LIN {X 0,Y 467.004,Z 300.757,A -85,B 0,C 180,E1 -6622.997,E2 -6622.997} C_VEL
LIN {X 0,Y 470.189,Z 309.996,A -85,B 0,C 180,E1 -6624.811,E2 -6624.811} C_VEL
LIN {X 0,Y 472.686,Z 318.668,A -85,B 0,C 180,E1 -6626.234,E2 -6626.234} C_VEL
LIN {X 0,Y 470.415,Z 339.223,A -85,B 0,C 180,E1 -6628.306,E2 -6628.306} C_VEL
LIN {X 0,Y 473.455,Z 359.975,A -85,B 0,C 180,E1 -6629.227,E2 -6629.227} C_VEL
LIN {X 0,Y 473.986,Z 366.788,A -85,B 0,C 180,E1 -6629.462,E2 -6629.462} C_VEL
LIN {X 0,Y 470.032,Z 462.753,A -85,B 0,C 180,E1 -6631.452,E2 -6631.452} C_VEL
LIN {X 0,Y 467.328,Z 564.491,A -85,B 0,C 180,E1 -6633.396,E2 -6633.396} C_VEL
LIN {X 0,Y 466.49,Z 584.331,A -85,B 0,C 180,E1 -6634.004,E2 -6634.004} C_VEL
LIN {X 0,Y 465.449,Z 603.573,A -85,B 0,C 180,E1 -6634.828,E2 -6634.828} C_VEL
LIN {X 0,Y 464.28,Z 621.738,A -85,B 0,C 180,E1 -6635.847,E2 -6635.847} C_VEL
LIN {X 0,Y 463.025,Z 638.947,A -85,B 0,C 180,E1 -6637.056,E2 -6637.056} C_VEL
LIN {X 0,Y 461.725,Z 655.288,A -85,B 0,C 180,E1 -6638.467,E2 -6638.467} C_VEL
LIN {X 0,Y 460.481,Z 669.969,A -85,B 0,C 180,E1 -6640.003,E2 -6640.003} C_VEL
LIN {X 0,Y 459.311,Z 683.717,A -85,B 0,C 180,E1 -6641.732,E2 -6641.732} C_VEL
LIN {X 0,Y 458.262,Z 696.374,A -85,B 0,C 180,E1 -6643.653,E2 -6643.653} C_VEL
LIN {X 0,Y 457.409,Z 707.461,A -85,B 0,C 180,E1 -6645.7,E2 -6645.7} C_VEL
LIN {X 0,Y 456.77,Z 717.003,A -85,B 0,C 180,E1 -6647.87,E2 -6647.87} C_VEL
LIN {X 0,Y 456.351,Z 724.573,A -85,B 0,C 180,E1 -6650.033,E2 -6650.033} C_VEL
LIN {X 0,Y 456.093,Z 730.779,A -85,B 0,C 180,E1 -6652.315,E2 -6652.315} C_VEL
LIN {X 0,Y 455.974,Z 735.448,A -85,B 0,C 180,E1 -6654.716,E2 -6654.716} C_VEL
LIN {X 0,Y 455.931,Z 738.322,A -85,B 0,C 180,E1 -6657.109,E2 -6657.109} C_VEL
LIN {X 0,Y 455.922,Z 739.49,A -85,B 0,C 180,E1 -6659.498,E2 -6659.498} C_VEL
LIN {X 0,Y 455.92,Z 739.024,A -85,B 0,C 180,E1 -6661.886,E2 -6661.886} C_VEL
LIN {X 0,Y 455.939,Z 736.915,A -85,B 0,C 180,E1 -6664.276,E2 -6664.276} C_VEL
LIN {X 0,Y 456.015,Z 733.052,A -85,B 0,C 180,E1 -6666.674,E2 -6666.674} C_VEL
LIN {X 0,Y 456.209,Z 727.319,A -85,B 0,C 180,E1 -6669.08,E2 -6669.08} C_VEL
LIN {X 0,Y 456.557,Z 720.008,A -85,B 0,C 180,E1 -6671.368,E2 -6671.368} C_VEL
LIN {X 0,Y 457.145,Z 710.687,A -85,B 0,C 180,E1 -6673.664,E2 -6673.664} C_VEL
LIN {X 0,Y 457.968,Z 699.685,A -85,B 0,C 180,E1 -6675.838,E2 -6675.838} C_VEL
LIN {X 0,Y 458.995,Z 687.344,A -85,B 0,C 180,E1 -6677.833,E2 -6677.833} C_VEL
LIN {X 0,Y 460.155,Z 674.019,A -85,B 0,C 180,E1 -6679.616,E2 -6679.616} C_VEL
LIN {X 0,Y 461.415,Z 659.738,A -85,B 0,C 180,E1 -6681.216,E2 -6681.216} C_VEL
LIN {X 0,Y 462.762,Z 643.878,A -85,B 0,C 180,E1 -6682.691,E2 -6682.691} C_VEL
LIN {X 0,Y 464.102,Z 627.202,A -85,B 0,C 180,E1 -6683.961,E2 -6683.961} C_VEL
LIN {X 0,Y 465.366,Z 609.596,A -85,B 0,C 180,E1 -6685.041,E2 -6685.041} C_VEL
LIN {X 0,Y 466.447,Z 591.759,A -85,B 0,C 180,E1 -6685.897,E2 -6685.897} C_VEL
LIN {X 0,Y 467.379,Z 572.839,A -85,B 0,C 180,E1 -6686.571,E2 -6686.571} C_VEL
LIN {X 0,Y 468.043,Z 553.455,A -85,B 0,C 180,E1 -6687.032,E2 -6687.032} C_VEL
LIN {X 0,Y 472.044,Z 364.66,A -85,B 0,C 180,E1 -6690.301,E2 -6690.301} C_VEL
LIN {X 0,Y 468.212,Z 340.667,A -85,B 0,C 180,E1 -6691.092,E2 -6691.092} C_VEL
LIN {X 0,Y 469.992,Z 315.315,A -85,B 0,C 180,E1 -6693.493,E2 -6693.493} C_VEL
LIN {X 0,Y 463.477,Z 296.548,A -85,B 0,C 180,E1 -6696.002,E2 -6696.002} C_VEL
LIN {X 0,Y 457.078,Z 279.761,A -85,B 0,C 180,E1 -6698.464,E2 -6698.464} C_VEL
LIN {X 0,Y 457.07,Z 279.544,A -85,B 0,C 180,E1 -6701.525,E2 -6701.525} C_VEL
LIN {X 0,Y 456.059,Z 279.675,A -85,B 0,C 180,E1 -6702.49,E2 -6702.49} C_VEL
LIN {X 0,Y 449.569,Z 280.487,A -85,B 0,C 180,E1 -6705.278,E2 -6705.278} C_VEL
LIN {X 0,Y 449.122,Z 280.541,A -85,B 0,C 180,E1 -6705.917,E2 -6705.917} C_VEL
LIN {X 0,Y 449.137,Z 280.538,A -85,B 0,C 180,E1 -6709.622,E2 -6709.622} C_VEL
LIN {X 0,Y 449.13,Z 280.537,A -85,B 0,C 180,E1 -6713.37,E2 -6713.37} C_VEL
LIN {X 0,Y 449.119,Z 280.539,A -85,B 0,C 180,E1 -6717.097,E2 -6717.097} C_VEL
LIN {X 0,Y 449.114,Z 280.527,A -85,B 0,C 180,E1 -6720.819,E2 -6720.819} C_VEL
LIN {X 0,Y 449.118,Z 280.528,A -85,B 0,C 180,E1 -6724.552,E2 -6724.552} C_VEL
LIN {X 0,Y 449.137,Z 280.53,A -85,B 0,C 180,E1 -6728.176,E2 -6728.176} C_VEL
LIN {X 0,Y 449.133,Z 280.53,A -85,B 0,C 180,E1 -6731.973,E2 -6731.973} C_VEL
LIN {X 0,Y 449.131,Z 280.608,A -85,B 0,C 180,E1 -6735.752,E2 -6735.752} C_VEL
LIN {X 0,Y 449.544,Z 282.242,A -85,B 0,C 180,E1 -6736.034,E2 -6736.034} C_VEL
LIN {X 0,Y 456.659,Z 302.01,A -85,B 0,C 180,E1 -6738.378,E2 -6738.378} C_VEL
LIN {X 0,Y 460.21,Z 313.576,A -85,B 0,C 180,E1 -6739.673,E2 -6739.673} C_VEL
LIN {X 0,Y 458.853,Z 354.962,A -85,B 0,C 180,E1 -6743.241,E2 -6743.241} C_VEL
LIN {X 0,Y 457.35,Z 396.302,A -85,B 0,C 180,E1 -6746.803,E2 -6746.803} C_VEL
LIN {X 0,Y 455.74,Z 437.908,A -85,B 0,C 180,E1 -6750.376,E2 -6750.376} C_VEL
LIN {X 0,Y 454.421,Z 476.738,A -85,B 0,C 180,E1 -6753.681,E2 -6753.681} C_VEL
LIN {X 0,Y 455.836,Z 490.567,A -85,B 0,C 180,E1 -6753.982,E2 -6753.982} C_VEL
LIN {X 0,Y 454.268,Z 619.633,A -85,B 0,C 180,E1 -6756.087,E2 -6756.087} C_VEL
LIN {X 0,Y 453.856,Z 635.661,A -85,B 0,C 180,E1 -6756.581,E2 -6756.581} C_VEL
LIN {X 0,Y 453.255,Z 650.989,A -85,B 0,C 180,E1 -6757.286,E2 -6757.286} C_VEL
LIN {X 0,Y 452.533,Z 665.232,A -85,B 0,C 180,E1 -6758.169,E2 -6758.169} C_VEL
LIN {X 0,Y 451.63,Z 679.94,A -85,B 0,C 180,E1 -6759.363,E2 -6759.363} C_VEL
LIN {X 0,Y 450.841,Z 692.096,A -85,B 0,C 180,E1 -6760.606,E2 -6760.606} C_VEL
LIN {X 0,Y 450.014,Z 704.083,A -85,B 0,C 180,E1 -6762.144,E2 -6762.144} C_VEL
LIN {X 0,Y 449.336,Z 714.291,A -85,B 0,C 180,E1 -6763.773,E2 -6763.773} C_VEL
LIN {X 0,Y 448.765,Z 723.452,A -85,B 0,C 180,E1 -6765.638,E2 -6765.638} C_VEL
LIN {X 0,Y 448.394,Z 730.619,A -85,B 0,C 180,E1 -6767.518,E2 -6767.518} C_VEL
LIN {X 0,Y 448.159,Z 736.252,A -85,B 0,C 180,E1 -6769.55,E2 -6769.55} C_VEL
LIN {X 0,Y 448.048,Z 740.095,A -85,B 0,C 180,E1 -6771.604,E2 -6771.604} C_VEL
LIN {X 0,Y 448.006,Z 742.118,A -85,B 0,C 180,E1 -6773.684,E2 -6773.684} C_VEL
LIN {X 0,Y 448.004,Z 742.42,A -85,B 0,C 180,E1 -6775.796,E2 -6775.796} C_VEL
LIN {X 0,Y 448.031,Z 741.006,A -85,B 0,C 180,E1 -6777.8,E2 -6777.8} C_VEL
LIN {X 0,Y 448.127,Z 737.586,A -85,B 0,C 180,E1 -6779.984,E2 -6779.984} C_VEL
LIN {X 0,Y 448.31,Z 732.813,A -85,B 0,C 180,E1 -6781.907,E2 -6781.907} C_VEL
LIN {X 0,Y 448.644,Z 726.109,A -85,B 0,C 180,E1 -6783.857,E2 -6783.857} C_VEL
LIN {X 0,Y 449.14,Z 717.93,A -85,B 0,C 180,E1 -6785.678,E2 -6785.678} C_VEL
LIN {X 0,Y 449.832,Z 707.5,A -85,B 0,C 180,E1 -6787.483,E2 -6787.483} C_VEL
LIN {X 0,Y 450.573,Z 696.876,A -85,B 0,C 180,E1 -6788.955,E2 -6788.955} C_VEL
LIN {X 0,Y 451.426,Z 684.129,A -85,B 0,C 180,E1 -6790.365,E2 -6790.365} C_VEL
LIN {X 0,Y 452.278,Z 670.794,A -85,B 0,C 180,E1 -6791.543,E2 -6791.543} C_VEL
LIN {X 0,Y 453.084,Z 656.003,A -85,B 0,C 180,E1 -6792.55,E2 -6792.55} C_VEL
LIN {X 0,Y 453.737,Z 641.285,A -85,B 0,C 180,E1 -6793.308,E2 -6793.308} C_VEL
LIN {X 0,Y 454.202,Z 625.159,A -85,B 0,C 180,E1 -6793.881,E2 -6793.881} C_VEL
LIN {X 0,Y 454.475,Z 607.28,A -85,B 0,C 180,E1 -6794.254,E2 -6794.254} C_VEL
LIN {X 0,Y 455.734,Z 487.115,A -85,B 0,C 180,E1 -6796.2,E2 -6796.2} C_VEL
LIN {X 0,Y 454.494,Z 476.284,A -85,B 0,C 180,E1 -6796.481,E2 -6796.481} C_VEL
LIN {X 0,Y 455.937,Z 434.163,A -85,B 0,C 180,E1 -6800.071,E2 -6800.071} C_VEL
LIN {X 0,Y 457.572,Z 390.761,A -85,B 0,C 180,E1 -6803.766,E2 -6803.766} C_VEL
LIN {X 0,Y 458.845,Z 346.921,A -85,B 0,C 180,E1 -6807.436,E2 -6807.436} C_VEL
LIN {X 0,Y 459.697,Z 311.528,A -85,B 0,C 180,E1 -6810.413,E2 -6810.413} C_VEL
LIN {X 0,Y 453.193,Z 291.764,A -85,B 0,C 180,E1 -6812.612,E2 -6812.612} C_VEL
LIN {X 0,Y 449.163,Z 280.91,A -85,B 0,C 180,E1 -6813.918,E2 -6813.918} C_VEL
LIN {X 0,Y 449.136,Z 280.536,A -85,B 0,C 180,E1 -6814.413,E2 -6814.413} C_VEL
LIN {X 0,Y 449.126,Z 280.539,A -85,B 0,C 180,E1 -6818.174,E2 -6818.174} C_VEL
LIN {X 0,Y 449.102,Z 280.536,A -85,B 0,C 180,E1 -6821.838,E2 -6821.838} C_VEL
LIN {X 0,Y 449.096,Z 280.541,A -85,B 0,C 180,E1 -6825.567,E2 -6825.567} C_VEL
LIN {X 0,Y 449.109,Z 280.539,A -85,B 0,C 180,E1 -6829.221,E2 -6829.221} C_VEL
LIN {X 0,Y 449.141,Z 280.537,A -85,B 0,C 180,E1 -6832.838,E2 -6832.838} C_VEL
LIN {X 0,Y 449.134,Z 280.54,A -85,B 0,C 180,E1 -6836.554,E2 -6836.554} C_VEL
LIN {X 0,Y 449.119,Z 280.544,A -85,B 0,C 180,E1 -6840.255,E2 -6840.255} C_VEL
LIN {X 0,Y 449.103,Z 280.539,A -85,B 0,C 180,E1 -6843.957,E2 -6843.957} C_VEL
LIN {X 0,Y 449.102,Z 280.539,A -85,B 0,C 180,E1 -6847.676,E2 -6847.676} C_VEL
LIN {X 0,Y 449.12,Z 280.538,A -85,B 0,C 180,E1 -6851.298,E2 -6851.298} C_VEL
LIN {X 0,Y 449.142,Z 280.535,A -85,B 0,C 180,E1 -6854.965,E2 -6854.965} C_VEL
LIN {X 0,Y 449.134,Z 280.537,A -85,B 0,C 180,E1 -6858.697,E2 -6858.697} C_VEL
LIN {X 0,Y 449.114,Z 280.538,A -85,B 0,C 180,E1 -6862.376,E2 -6862.376} C_VEL
LIN {X 0,Y 449.104,Z 280.541,A -85,B 0,C 180,E1 -6866.013,E2 -6866.013} C_VEL
LIN {X 0,Y 449.11,Z 280.536,A -85,B 0,C 180,E1 -6869.766,E2 -6869.766} C_VEL
LIN {X 0,Y 449.133,Z 280.537,A -85,B 0,C 180,E1 -6873.406,E2 -6873.406} C_VEL
LIN {X 0,Y 449.139,Z 280.538,A -85,B 0,C 180,E1 -6877.162,E2 -6877.162} C_VEL
LIN {X 0,Y 449.139,Z 280.54,A -85,B 0,C 180,E1 -6880.881,E2 -6880.881} C_VEL
LIN {X 0,Y 449.119,Z 280.541,A -85,B 0,C 180,E1 -6884.572,E2 -6884.572} C_VEL
LIN {X 0,Y 449.141,Z 280.773,A -85,B 0,C 180,E1 -6888.078,E2 -6888.078} C_VEL
LIN {X 0,Y 451.649,Z 287.077,A -85,B 0,C 180,E1 -6889.017,E2 -6889.017} C_VEL
LIN {X 0,Y 460.318,Z 307.995,A -85,B 0,C 180,E1 -6891.841,E2 -6891.841} C_VEL
LIN {X 0,Y 463.887,Z 317.307,A -85,B 0,C 180,E1 -6892.994,E2 -6892.994} C_VEL
LIN {X 0,Y 467.002,Z 323.829,A -85,B 0,C 180,E1 -6893.412,E2 -6893.412} C_VEL
LIN {X 0,Y 469.493,Z 342.184,A -85,B 0,C 180,E1 -6893.988,E2 -6893.988} C_VEL
LIN {X 0,Y 464.853,Z 535.757,A -85,B 0,C 180,E1 -6897.4,E2 -6897.4} C_VEL
LIN {X 0,Y 463.81,Z 578.935,A -85,B 0,C 180,E1 -6898.185,E2 -6898.185} C_VEL
LIN {X 0,Y 462.812,Z 599.678,A -85,B 0,C 180,E1 -6898.776,E2 -6898.776} C_VEL
LIN {X 0,Y 461.518,Z 620.38,A -85,B 0,C 180,E1 -6899.606,E2 -6899.606} C_VEL
LIN {X 0,Y 460.009,Z 640.141,A -85,B 0,C 180,E1 -6900.644,E2 -6900.644} C_VEL
LIN {X 0,Y 458.457,Z 658.206,A -85,B 0,C 180,E1 -6901.827,E2 -6901.827} C_VEL
LIN {X 0,Y 456.739,Z 676.474,A -85,B 0,C 180,E1 -6903.273,E2 -6903.273} C_VEL
LIN {X 0,Y 454.965,Z 694.499,A -85,B 0,C 180,E1 -6904.994,E2 -6904.994} C_VEL
LIN {X 0,Y 453.312,Z 711.029,A -85,B 0,C 180,E1 -6906.885,E2 -6906.885} C_VEL
LIN {X 0,Y 451.875,Z 725.61,A -85,B 0,C 180,E1 -6908.861,E2 -6908.861} C_VEL
LIN {X 0,Y 450.656,Z 738.782,A -85,B 0,C 180,E1 -6910.967,E2 -6910.967} C_VEL
LIN {X 0,Y 449.621,Z 751.154,A -85,B 0,C 180,E1 -6913.331,E2 -6913.331} C_VEL
LIN {X 0,Y 448.858,Z 761.842,A -85,B 0,C 180,E1 -6915.818,E2 -6915.818} C_VEL
LIN {X 0,Y 448.37,Z 770.416,A -85,B 0,C 180,E1 -6918.293,E2 -6918.293} C_VEL
LIN {X 0,Y 448.097,Z 777.147,A -85,B 0,C 180,E1 -6920.757,E2 -6920.757} C_VEL
LIN {X 0,Y 447.976,Z 782.424,A -85,B 0,C 180,E1 -6923.337,E2 -6923.337} C_VEL
LIN {X 0,Y 447.934,Z 785.83,A -85,B 0,C 180,E1 -6925.777,E2 -6925.777} C_VEL
LIN {X 0,Y 447.924,Z 787.706,A -85,B 0,C 180,E1 -6928.339,E2 -6928.339} C_VEL
LIN {X 0,Y 447.93,Z 787.934,A -85,B 0,C 180,E1 -6930.769,E2 -6930.769} C_VEL
LIN {X 0,Y 447.924,Z 786.591,A -85,B 0,C 180,E1 -6933.329,E2 -6933.329} C_VEL
LIN {X 0,Y 447.954,Z 783.781,A -85,B 0,C 180,E1 -6935.766,E2 -6935.766} C_VEL
LIN {X 0,Y 448.055,Z 779.035,A -85,B 0,C 180,E1 -6938.342,E2 -6938.342} C_VEL
LIN {X 0,Y 448.26,Z 772.794,A -85,B 0,C 180,E1 -6940.8,E2 -6940.8} C_VEL
LIN {X 0,Y 448.64,Z 764.715,A -85,B 0,C 180,E1 -6943.272,E2 -6943.272} C_VEL
LIN {X 0,Y 449.278,Z 754.556,A -85,B 0,C 180,E1 -6945.755,E2 -6945.755} C_VEL
LIN {X 0,Y 450.13,Z 743.005,A -85,B 0,C 180,E1 -6948.067,E2 -6948.067} C_VEL
LIN {X 0,Y 451.188,Z 730.06,A -85,B 0,C 180,E1 -6950.226,E2 -6950.226} C_VEL
LIN {X 0,Y 452.465,Z 715.399,A -85,B 0,C 180,E1 -6952.272,E2 -6952.272} C_VEL
LIN {X 0,Y 453.839,Z 699.789,A -85,B 0,C 180,E1 -6954.103,E2 -6954.103} C_VEL
LIN {X 0,Y 455.316,Z 682.894,A -85,B 0,C 180,E1 -6955.774,E2 -6955.774} C_VEL
LIN {X 0,Y 456.751,Z 665.337,A -85,B 0,C 180,E1 -6957.228,E2 -6957.228} C_VEL
LIN {X 0,Y 458.24,Z 646.072,A -85,B 0,C 180,E1 -6958.546,E2 -6958.546} C_VEL
LIN {X 0,Y 459.606,Z 625.931,A -85,B 0,C 180,E1 -6959.656,E2 -6959.656} C_VEL
LIN {X 0,Y 460.785,Z 605.455,A -85,B 0,C 180,E1 -6960.534,E2 -6960.534} C_VEL
LIN {X 0,Y 461.742,Z 584.721,A -85,B 0,C 180,E1 -6961.188,E2 -6961.188} C_VEL
LIN {X 0,Y 462.403,Z 562.319,A -85,B 0,C 180,E1 -6961.658,E2 -6961.658} C_VEL
LIN {X 0,Y 464.451,Z 466.12,A -85,B 0,C 180,E1 -6963.371,E2 -6963.371} C_VEL
LIN {X 0,Y 467.579,Z 374.807,A -85,B 0,C 180,E1 -6965.199,E2 -6965.199} C_VEL
LIN {X 0,Y 468.939,Z 339.731,A -85,B 0,C 180,E1 -6965.974,E2 -6965.974} C_VEL
LIN {X 0,Y 467.087,Z 323.355,A -85,B 0,C 180,E1 -6966.634,E2 -6966.634} C_VEL
LIN {X 0,Y 466.104,Z 320.719,A -85,B 0,C 180,E1 -6966.917,E2 -6966.917} C_VEL
LIN {X 0,Y 463.19,Z 310.793,A -85,B 0,C 180,E1 -6968.51,E2 -6968.51} C_VEL
LIN {X 0,Y 460.486,Z 303.252,A -85,B 0,C 180,E1 -6970.049,E2 -6970.049} C_VEL
LIN {X 0,Y 458.316,Z 298.482,A -85,B 0,C 180,E1 -6971.379,E2 -6971.379} C_VEL
LIN {X 0,Y 456.97,Z 295.312,A -85,B 0,C 180,E1 -6972.493,E2 -6972.493} C_VEL
LIN {X 0,Y 455.479,Z 292.157,A -85,B 0,C 180,E1 -6974.306,E2 -6974.306} C_VEL
LIN {X 0,Y 455.145,Z 291.254,A -85,B 0,C 180,E1 -6975.379,E2 -6975.379} C_VEL
LIN {X 0,Y 455.306,Z 291.516,A -85,B 0,C 180,E1 -6977.097,E2 -6977.097} C_VEL
LIN {X 0,Y 456.358,Z 294.584,A -85,B 0,C 180,E1 -6979.103,E2 -6979.103} C_VEL
LIN {X 0,Y 457.325,Z 296.299,A -85,B 0,C 180,E1 -6979.927,E2 -6979.927} C_VEL
LIN {X 0,Y 458.999,Z 300.428,A -85,B 0,C 180,E1 -6981.305,E2 -6981.305} C_VEL
LIN {X 0,Y 461.244,Z 306.052,A -85,B 0,C 180,E1 -6982.786,E2 -6982.786} C_VEL
LIN {X 0,Y 464.121,Z 314.873,A -85,B 0,C 180,E1 -6984.584,E2 -6984.584} C_VEL
LIN {X 0,Y 466.083,Z 322.779,A -85,B 0,C 180,E1 -6985.901,E2 -6985.901} C_VEL
LIN {X 0,Y 464.085,Z 338.535,A -85,B 0,C 180,E1 -6987.539,E2 -6987.539} C_VEL
LIN {X 0,Y 466.875,Z 358.34,A -85,B 0,C 180,E1 -6988.493,E2 -6988.493} C_VEL
LIN {X 0,Y 467.732,Z 367.877,A -85,B 0,C 180,E1 -6988.866,E2 -6988.866} C_VEL
LIN {X 0,Y 463.358,Z 459.298,A -85,B 0,C 180,E1 -6990.861,E2 -6990.861} C_VEL
LIN {X 0,Y 460.584,Z 549.83,A -85,B 0,C 180,E1 -6992.649,E2 -6992.649} C_VEL
LIN {X 0,Y 459.83,Z 571.487,A -85,B 0,C 180,E1 -6993.154,E2 -6993.154} C_VEL
LIN {X 0,Y 458.842,Z 591.186,A -85,B 0,C 180,E1 -6993.854,E2 -6993.854} C_VEL
LIN {X 0,Y 457.656,Z 610.428,A -85,B 0,C 180,E1 -6994.785,E2 -6994.785} C_VEL
LIN {X 0,Y 456.377,Z 628.154,A -85,B 0,C 180,E1 -6995.884,E2 -6995.884} C_VEL
LIN {X 0,Y 455.03,Z 644.916,A -85,B 0,C 180,E1 -6997.17,E2 -6997.17} C_VEL
LIN {X 0,Y 453.711,Z 660.341,A -85,B 0,C 180,E1 -6998.61,E2 -6998.61} C_VEL
LIN {X 0,Y 452.418,Z 674.823,A -85,B 0,C 180,E1 -7000.237,E2 -7000.237} C_VEL
LIN {X 0,Y 451.209,Z 688.298,A -85,B 0,C 180,E1 -7002.061,E2 -7002.061} C_VEL
LIN {X 0,Y 450.168,Z 700.262,A -85,B 0,C 180,E1 -7004.014,E2 -7004.014} C_VEL
LIN {X 0,Y 449.334,Z 710.752,A -85,B 0,C 180,E1 -7006.095,E2 -7006.095} C_VEL
LIN {X 0,Y 448.713,Z 719.754,A -85,B 0,C 180,E1 -7008.301,E2 -7008.301} C_VEL
LIN {X 0,Y 448.319,Z 726.882,A -85,B 0,C 180,E1 -7010.501,E2 -7010.501} C_VEL
LIN {X 0,Y 448.084,Z 732.617,A -85,B 0,C 180,E1 -7012.822,E2 -7012.822} C_VEL
LIN {X 0,Y 447.975,Z 736.798,A -85,B 0,C 180,E1 -7015.263,E2 -7015.263} C_VEL
LIN {X 0,Y 447.941,Z 739.228,A -85,B 0,C 180,E1 -7017.698,E2 -7017.698} C_VEL
LIN {X 0,Y 447.94,Z 739.996,A -85,B 0,C 180,E1 -7020.128,E2 -7020.128} C_VEL
LIN {X 0,Y 447.94,Z 739.07,A -85,B 0,C 180,E1 -7022.559,E2 -7022.559} C_VEL
LIN {X 0,Y 447.974,Z 736.442,A -85,B 0,C 180,E1 -7024.994,E2 -7024.994} C_VEL
LIN {X 0,Y 448.088,Z 732.064,A -85,B 0,C 180,E1 -7027.437,E2 -7027.437} C_VEL
LIN {X 0,Y 448.35,Z 725.79,A -85,B 0,C 180,E1 -7029.888,E2 -7029.888} C_VEL
LIN {X 0,Y 448.796,Z 717.917,A -85,B 0,C 180,E1 -7032.219,E2 -7032.219} C_VEL
LIN {X 0,Y 449.462,Z 708.514,A -85,B 0,C 180,E1 -7034.428,E2 -7034.428} C_VEL
LIN {X 0,Y 450.354,Z 697.621,A -85,B 0,C 180,E1 -7036.51,E2 -7036.51} C_VEL
LIN {X 0,Y 451.46,Z 685.251,A -85,B 0,C 180,E1 -7038.464,E2 -7038.464} C_VEL
LIN {X 0,Y 452.754,Z 671.351,A -85,B 0,C 180,E1 -7040.287,E2 -7040.287} C_VEL
LIN {X 0,Y 454.128,Z 656.651,A -85,B 0,C 180,E1 -7041.892,E2 -7041.892} C_VEL
LIN {X 0,Y 455.557,Z 640.643,A -85,B 0,C 180,E1 -7043.339,E2 -7043.339} C_VEL
LIN {X 0,Y 456.934,Z 624.078,A -85,B 0,C 180,E1 -7044.568,E2 -7044.568} C_VEL
LIN {X 0,Y 458.211,Z 606.847,A -85,B 0,C 180,E1 -7045.599,E2 -7045.599} C_VEL
LIN {X 0,Y 459.404,Z 587.701,A -85,B 0,C 180,E1 -7046.481,E2 -7046.481} C_VEL
LIN {X 0,Y 460.322,Z 568.448,A -85,B 0,C 180,E1 -7047.124,E2 -7047.124} C_VEL
LIN {X 0,Y 460.979,Z 547.683,A -85,B 0,C 180,E1 -7047.57,E2 -7047.57} C_VEL
LIN {X 0,Y 465.162,Z 367.88,A -85,B 0,C 180,E1 -7050.755,E2 -7050.755} C_VEL
LIN {X 0,Y 464.681,Z 362.556,A -85,B 0,C 180,E1 -7050.899,E2 -7050.899} C_VEL
LIN {X 0,Y 461.179,Z 340.621,A -85,B 0,C 180,E1 -7051.647,E2 -7051.647} C_VEL
LIN {X 0,Y 462.937,Z 318.632,A -85,B 0,C 180,E1 -7053.743,E2 -7053.743} C_VEL
LIN {X 0,Y 456.59,Z 300.164,A -85,B 0,C 180,E1 -7056.247,E2 -7056.247} C_VEL
LIN {X 0,Y 449.169,Z 280.738,A -85,B 0,C 180,E1 -7059.135,E2 -7059.135} C_VEL
LIN {X 0,Y 449.133,Z 280.54,A -85,B 0,C 180,E1 -7062.766,E2 -7062.766} C_VEL
LIN {X 0,Y 449.122,Z 280.541,A -85,B 0,C 180,E1 -7065.917,E2 -7065.917} C_VEL
LIN {X 0,Y 448.112,Z 280.666,A -85,B 0,C 180,E1 -7066.899,E2 -7066.899} C_VEL
LIN {X 0,Y 441.609,Z 281.477,A -85,B 0,C 180,E1 -7069.738,E2 -7069.738} C_VEL
LIN {X 0,Y 441.192,Z 281.529,A -85,B 0,C 180,E1 -7070.388,E2 -7070.388} C_VEL
LIN {X 0,Y 441.191,Z 281.529,A -85,B 0,C 180,E1 -7074.227,E2 -7074.227} C_VEL
LIN {X 0,Y 441.198,Z 281.527,A -85,B 0,C 180,E1 -7077.973,E2 -7077.973} C_VEL
LIN {X 0,Y 441.199,Z 281.519,A -85,B 0,C 180,E1 -7081.728,E2 -7081.728} C_VEL
LIN {X 0,Y 441.18,Z 281.517,A -85,B 0,C 180,E1 -7085.496,E2 -7085.496} C_VEL
LIN {X 0,Y 441.158,Z 281.522,A -85,B 0,C 180,E1 -7089.154,E2 -7089.154} C_VEL
LIN {X 0,Y 441.149,Z 281.531,A -85,B 0,C 180,E1 -7092.863,E2 -7092.863} C_VEL
LIN {X 0,Y 441.173,Z 281.72,A -85,B 0,C 180,E1 -7095.227,E2 -7095.227} C_VEL
LIN {X 0,Y 442.32,Z 284.77,A -85,B 0,C 180,E1 -7095.668,E2 -7095.668} C_VEL
LIN {X 0,Y 450.223,Z 307.11,A -85,B 0,C 180,E1 -7098.347,E2 -7098.347} C_VEL
LIN {X 0,Y 452.973,Z 316.25,A -85,B 0,C 180,E1 -7099.378,E2 -7099.378} C_VEL
LIN {X 0,Y 451.506,Z 357.126,A -85,B 0,C 180,E1 -7102.939,E2 -7102.939} C_VEL
LIN {X 0,Y 449.934,Z 398.081,A -85,B 0,C 180,E1 -7106.495,E2 -7106.495} C_VEL
LIN {X 0,Y 448.236,Z 439.173,A -85,B 0,C 180,E1 -7110.063,E2 -7110.063} C_VEL
LIN {X 0,Y 446.887,Z 477.018,A -85,B 0,C 180,E1 -7113.309,E2 -7113.309} C_VEL
LIN {X 0,Y 448.356,Z 491.357,A -85,B 0,C 180,E1 -7113.631,E2 -7113.631} C_VEL
LIN {X 0,Y 446.695,Z 620.089,A -85,B 0,C 180,E1 -7115.763,E2 -7115.763} C_VEL
LIN {X 0,Y 446.261,Z 636.081,A -85,B 0,C 180,E1 -7116.265,E2 -7116.265} C_VEL
LIN {X 0,Y 445.592,Z 652.169,A -85,B 0,C 180,E1 -7117.023,E2 -7117.023} C_VEL
LIN {X 0,Y 444.806,Z 666.508,A -85,B 0,C 180,E1 -7117.945,E2 -7117.945} C_VEL
LIN {X 0,Y 443.877,Z 680.803,A -85,B 0,C 180,E1 -7119.136,E2 -7119.136} C_VEL
LIN {X 0,Y 442.998,Z 693.41,A -85,B 0,C 180,E1 -7120.467,E2 -7120.467} C_VEL
LIN {X 0,Y 442.144,Z 705.063,A -85,B 0,C 180,E1 -7122.006,E2 -7122.006} C_VEL
LIN {X 0,Y 441.429,Z 715.121,A -85,B 0,C 180,E1 -7123.659,E2 -7123.659} C_VEL
LIN {X 0,Y 440.834,Z 724.039,A -85,B 0,C 180,E1 -7125.522,E2 -7125.522} C_VEL
LIN {X 0,Y 440.434,Z 731.159,A -85,B 0,C 180,E1 -7127.436,E2 -7127.436} C_VEL
LIN {X 0,Y 440.181,Z 736.749,A -85,B 0,C 180,E1 -7129.504,E2 -7129.504} C_VEL
LIN {X 0,Y 440.061,Z 740.552,A -85,B 0,C 180,E1 -7131.595,E2 -7131.595} C_VEL
LIN {X 0,Y 440.015,Z 742.533,A -85,B 0,C 180,E1 -7133.714,E2 -7133.714} C_VEL
LIN {X 0,Y 440.014,Z 742.803,A -85,B 0,C 180,E1 -7135.865,E2 -7135.865} C_VEL
LIN {X 0,Y 440.046,Z 741.335,A -85,B 0,C 180,E1 -7137.907,E2 -7137.907} C_VEL
LIN {X 0,Y 440.151,Z 738.009,A -85,B 0,C 180,E1 -7140.06,E2 -7140.06} C_VEL
LIN {X 0,Y 440.36,Z 733.034,A -85,B 0,C 180,E1 -7142.092,E2 -7142.092} C_VEL
LIN {X 0,Y 440.738,Z 726.189,A -85,B 0,C 180,E1 -7144.101,E2 -7144.101} C_VEL
LIN {X 0,Y 441.277,Z 718.01,A -85,B 0,C 180,E1 -7145.931,E2 -7145.931} C_VEL
LIN {X 0,Y 442.008,Z 707.793,A -85,B 0,C 180,E1 -7147.724,E2 -7147.724} C_VEL
LIN {X 0,Y 442.843,Z 696.61,A -85,B 0,C 180,E1 -7149.285,E2 -7149.285} C_VEL
LIN {X 0,Y 443.748,Z 683.902,A -85,B 0,C 180,E1 -7150.701,E2 -7150.701} C_VEL
LIN {X 0,Y 444.656,Z 670.333,A -85,B 0,C 180,E1 -7151.901,E2 -7151.901} C_VEL
LIN {X 0,Y 445.545,Z 654.948,A -85,B 0,C 180,E1 -7152.947,E2 -7152.947} C_VEL
LIN {X 0,Y 446.221,Z 639.636,A -85,B 0,C 180,E1 -7153.716,E2 -7153.716} C_VEL
LIN {X 0,Y 446.712,Z 622.753,A -85,B 0,C 180,E1 -7154.291,E2 -7154.291} C_VEL
LIN {X 0,Y 447.044,Z 598.324,A -85,B 0,C 180,E1 -7154.744,E2 -7154.744} C_VEL
LIN {X 0,Y 448.29,Z 488.008,A -85,B 0,C 180,E1 -7156.56,E2 -7156.56} C_VEL
LIN {X 0,Y 447.015,Z 476.916,A -85,B 0,C 180,E1 -7156.848,E2 -7156.848} C_VEL
LIN {X 0,Y 448.557,Z 433.644,A -85,B 0,C 180,E1 -7160.558,E2 -7160.558} C_VEL
LIN {X 0,Y 450.183,Z 391.513,A -85,B 0,C 180,E1 -7164.158,E2 -7164.158} C_VEL
LIN {X 0,Y 451.444,Z 352.894,A -85,B 0,C 180,E1 -7167.438,E2 -7167.438} C_VEL
LIN {X 0,Y 452.462,Z 314.159,A -85,B 0,C 180,E1 -7170.73,E2 -7170.73} C_VEL
LIN {X 0,Y 446.407,Z 295.705,A -85,B 0,C 180,E1 -7172.811,E2 -7172.811} C_VEL
LIN {X 0,Y 441.254,Z 281.906,A -85,B 0,C 180,E1 -7174.498,E2 -7174.498} C_VEL
LIN {X 0,Y 441.178,Z 281.529,A -85,B 0,C 180,E1 -7174.924,E2 -7174.924} C_VEL
LIN {X 0,Y 441.198,Z 281.522,A -85,B 0,C 180,E1 -7178.652,E2 -7178.652} C_VEL
LIN {X 0,Y 441.197,Z 281.527,A -85,B 0,C 180,E1 -7182.457,E2 -7182.457} C_VEL
LIN {X 0,Y 441.185,Z 281.533,A -85,B 0,C 180,E1 -7186.233,E2 -7186.233} C_VEL
LIN {X 0,Y 441.166,Z 281.531,A -85,B 0,C 180,E1 -7189.949,E2 -7189.949} C_VEL
LIN {X 0,Y 441.16,Z 281.529,A -85,B 0,C 180,E1 -7193.623,E2 -7193.623} C_VEL
LIN {X 0,Y 441.167,Z 281.529,A -85,B 0,C 180,E1 -7197.402,E2 -7197.402} C_VEL
LIN {X 0,Y 441.191,Z 281.524,A -85,B 0,C 180,E1 -7201.038,E2 -7201.038} C_VEL
LIN {X 0,Y 441.199,Z 281.529,A -85,B 0,C 180,E1 -7204.809,E2 -7204.809} C_VEL
LIN {X 0,Y 441.196,Z 281.528,A -85,B 0,C 180,E1 -7208.602,E2 -7208.602} C_VEL
LIN {X 0,Y 441.18,Z 281.528,A -85,B 0,C 180,E1 -7212.379,E2 -7212.379} C_VEL
LIN {X 0,Y 441.166,Z 281.526,A -85,B 0,C 180,E1 -7216.072,E2 -7216.072} C_VEL
LIN {X 0,Y 441.164,Z 281.528,A -85,B 0,C 180,E1 -7219.874,E2 -7219.874} C_VEL
LIN {X 0,Y 441.173,Z 281.528,A -85,B 0,C 180,E1 -7223.649,E2 -7223.649} C_VEL
LIN {X 0,Y 441.191,Z 281.525,A -85,B 0,C 180,E1 -7227.39,E2 -7227.39} C_VEL
LIN {X 0,Y 441.201,Z 281.527,A -85,B 0,C 180,E1 -7231.111,E2 -7231.111} C_VEL
LIN {X 0,Y 441.198,Z 281.531,A -85,B 0,C 180,E1 -7234.881,E2 -7234.881} C_VEL
LIN {X 0,Y 441.192,Z 281.531,A -85,B 0,C 180,E1 -7238.718,E2 -7238.718} C_VEL
LIN {X 0,Y 441.177,Z 281.532,A -85,B 0,C 180,E1 -7242.482,E2 -7242.482} C_VEL
LIN {X 0,Y 441.171,Z 281.531,A -85,B 0,C 180,E1 -7246.274,E2 -7246.274} C_VEL
LIN {X 0,Y 441.247,Z 281.87,A -85,B 0,C 180,E1 -7247.382,E2 -7247.382} C_VEL
LIN {X 0,Y 450.274,Z 303.715,A -85,B 0,C 180,E1 -7250.501,E2 -7250.501} C_VEL
LIN {X 0,Y 455.991,Z 317.99,A -85,B 0,C 180,E1 -7252.332,E2 -7252.332} C_VEL
LIN {X 0,Y 460.666,Z 327.189,A -85,B 0,C 180,E1 -7252.944,E2 -7252.944} C_VEL
LIN {X 0,Y 462.807,Z 343.497,A -85,B 0,C 180,E1 -7253.462,E2 -7253.462} C_VEL
LIN {X 0,Y 457.811,Z 535.941,A -85,B 0,C 180,E1 -7256.928,E2 -7256.928} C_VEL
LIN {X 0,Y 456.712,Z 578.69,A -85,B 0,C 180,E1 -7257.719,E2 -7257.719} C_VEL
LIN {X 0,Y 455.661,Z 599.497,A -85,B 0,C 180,E1 -7258.321,E2 -7258.321} C_VEL
LIN {X 0,Y 454.252,Z 620.653,A -85,B 0,C 180,E1 -7259.184,E2 -7259.184} C_VEL
LIN {X 0,Y 452.631,Z 640.786,A -85,B 0,C 180,E1 -7260.264,E2 -7260.264} C_VEL
LIN {X 0,Y 450.918,Z 659.614,A -85,B 0,C 180,E1 -7261.529,E2 -7261.529} C_VEL
LIN {X 0,Y 449.126,Z 677.545,A -85,B 0,C 180,E1 -7262.992,E2 -7262.992} C_VEL
LIN {X 0,Y 447.343,Z 694.663,A -85,B 0,C 180,E1 -7264.666,E2 -7264.666} C_VEL
LIN {X 0,Y 445.58,Z 711.241,A -85,B 0,C 180,E1 -7266.602,E2 -7266.602} C_VEL
LIN {X 0,Y 444.067,Z 725.727,A -85,B 0,C 180,E1 -7268.609,E2 -7268.609} C_VEL
LIN {X 0,Y 442.781,Z 738.828,A -85,B 0,C 180,E1 -7270.752,E2 -7270.752} C_VEL
LIN {X 0,Y 441.743,Z 750.531,A -85,B 0,C 180,E1 -7273.025,E2 -7273.025} C_VEL
LIN {X 0,Y 440.958,Z 760.738,A -85,B 0,C 180,E1 -7275.424,E2 -7275.424} C_VEL
LIN {X 0,Y 440.444,Z 769.059,A -85,B 0,C 180,E1 -7277.814,E2 -7277.814} C_VEL
LIN {X 0,Y 440.125,Z 776.357,A -85,B 0,C 180,E1 -7280.456,E2 -7280.456} C_VEL
LIN {X 0,Y 439.984,Z 781.551,A -85,B 0,C 180,E1 -7282.953,E2 -7282.953} C_VEL
LIN {X 0,Y 439.941,Z 785.113,A -85,B 0,C 180,E1 -7285.439,E2 -7285.439} C_VEL
LIN {X 0,Y 439.94,Z 787.077,A -85,B 0,C 180,E1 -7287.918,E2 -7287.918} C_VEL
LIN {X 0,Y 439.937,Z 787.552,A -85,B 0,C 180,E1 -7290.522,E2 -7290.522} C_VEL
LIN {X 0,Y 439.937,Z 786.489,A -85,B 0,C 180,E1 -7292.998,E2 -7292.998} C_VEL
LIN {X 0,Y 439.952,Z 783.805,A -85,B 0,C 180,E1 -7295.487,E2 -7295.487} C_VEL
LIN {X 0,Y 440.044,Z 779.312,A -85,B 0,C 180,E1 -7298.1,E2 -7298.1} C_VEL
LIN {X 0,Y 440.252,Z 772.933,A -85,B 0,C 180,E1 -7300.734,E2 -7300.734} C_VEL
LIN {X 0,Y 440.634,Z 764.984,A -85,B 0,C 180,E1 -7303.25,E2 -7303.25} C_VEL
LIN {X 0,Y 441.243,Z 755.554,A -85,B 0,C 180,E1 -7305.645,E2 -7305.645} C_VEL
LIN {X 0,Y 442.122,Z 743.965,A -85,B 0,C 180,E1 -7308.05,E2 -7308.05} C_VEL
LIN {X 0,Y 443.172,Z 731.504,A -85,B 0,C 180,E1 -7310.195,E2 -7310.195} C_VEL
LIN {X 0,Y 444.435,Z 717.672,A -85,B 0,C 180,E1 -7312.208,E2 -7312.208} C_VEL
LIN {X 0,Y 445.876,Z 702.126,A -85,B 0,C 180,E1 -7314.122,E2 -7314.122} C_VEL
LIN {X 0,Y 447.474,Z 684.889,A -85,B 0,C 180,E1 -7315.903,E2 -7315.903} C_VEL
LIN {X 0,Y 449.047,Z 666.984,A -85,B 0,C 180,E1 -7317.447,E2 -7317.447} C_VEL
LIN {X 0,Y 450.605,Z 648.2,A -85,B 0,C 180,E1 -7318.785,E2 -7318.785} C_VEL
LIN {X 0,Y 452.045,Z 628.603,A -85,B 0,C 180,E1 -7319.92,E2 -7319.92} C_VEL
LIN {X 0,Y 453.369,Z 607.681,A -85,B 0,C 180,E1 -7320.867,E2 -7320.867} C_VEL
LIN {X 0,Y 454.47,Z 585.842,A -85,B 0,C 180,E1 -7321.593,E2 -7321.593} C_VEL
LIN {X 0,Y 455.219,Z 563.267,A -85,B 0,C 180,E1 -7322.088,E2 -7322.088} C_VEL
LIN {X 0,Y 457.443,Z 471.715,A -85,B 0,C 180,E1 -7323.781,E2 -7323.781} C_VEL
LIN {X 0,Y 460.734,Z 385.677,A -85,B 0,C 180,E1 -7325.569,E2 -7325.569} C_VEL
LIN {X 0,Y 462.815,Z 341.137,A -85,B 0,C 180,E1 -7326.591,E2 -7326.591} C_VEL
LIN {X 0,Y 461.409,Z 327.079,A -85,B 0,C 180,E1 -7327.193,E2 -7327.193} C_VEL
LIN {X 0,Y 459.208,Z 322.242,A -85,B 0,C 180,E1 -7327.678,E2 -7327.678} C_VEL
LIN {X 0,Y 456.915,Z 314.351,A -85,B 0,C 180,E1 -7329.068,E2 -7329.068} C_VEL
LIN {X 0,Y 454.658,Z 308.19,A -85,B 0,C 180,E1 -7330.457,E2 -7330.457} C_VEL
LIN {X 0,Y 453.091,Z 304.346,A -85,B 0,C 180,E1 -7331.575,E2 -7331.575} C_VEL
LIN {X 0,Y 451.999,Z 301.525,A -85,B 0,C 180,E1 -7332.603,E2 -7332.603} C_VEL
LIN {X 0,Y 450.664,Z 298.499,A -85,B 0,C 180,E1 -7334.406,E2 -7334.406} C_VEL
LIN {X 0,Y 450.382,Z 297.678,A -85,B 0,C 180,E1 -7335.451,E2 -7335.451} C_VEL
LIN {X 0,Y 450.505,Z 297.961,A -85,B 0,C 180,E1 -7337.09,E2 -7337.09} C_VEL
LIN {X 0,Y 451.405,Z 300.859,A -85,B 0,C 180,E1 -7339.054,E2 -7339.054} C_VEL
LIN {X 0,Y 452.242,Z 302.678,A -85,B 0,C 180,E1 -7339.905,E2 -7339.905} C_VEL
LIN {X 0,Y 453.759,Z 306.663,A -85,B 0,C 180,E1 -7341.265,E2 -7341.265} C_VEL
LIN {X 0,Y 455.605,Z 311.582,A -85,B 0,C 180,E1 -7342.603,E2 -7342.603} C_VEL
LIN {X 0,Y 458.153,Z 319.894,A -85,B 0,C 180,E1 -7344.36,E2 -7344.36} C_VEL
LIN {X 0,Y 459.651,Z 326.416,A -85,B 0,C 180,E1 -7345.491,E2 -7345.491} C_VEL
LIN {X 0,Y 458.028,Z 338.193,A -85,B 0,C 180,E1 -7346.739,E2 -7346.739} C_VEL
LIN {X 0,Y 460.688,Z 358.394,A -85,B 0,C 180,E1 -7347.792,E2 -7347.792} C_VEL
LIN {X 0,Y 461.626,Z 369.193,A -85,B 0,C 180,E1 -7348.243,E2 -7348.243} C_VEL
LIN {X 0,Y 456.809,Z 456.691,A -85,B 0,C 180,E1 -7350.249,E2 -7350.249} C_VEL
LIN {X 0,Y 453.689,Z 542.646,A -85,B 0,C 180,E1 -7352.044,E2 -7352.044} C_VEL
LIN {X 0,Y 452.772,Z 568.529,A -85,B 0,C 180,E1 -7352.622,E2 -7352.622} C_VEL
LIN {X 0,Y 451.765,Z 588.323,A -85,B 0,C 180,E1 -7353.303,E2 -7353.303} C_VEL
LIN {X 0,Y 450.577,Z 606.905,A -85,B 0,C 180,E1 -7354.172,E2 -7354.172} C_VEL
LIN {X 0,Y 449.224,Z 625.06,A -85,B 0,C 180,E1 -7355.264,E2 -7355.264} C_VEL
LIN {X 0,Y 447.734,Z 642.969,A -85,B 0,C 180,E1 -7356.612,E2 -7356.612} C_VEL
LIN {X 0,Y 446.223,Z 659.644,A -85,B 0,C 180,E1 -7358.164,E2 -7358.164} C_VEL
LIN {X 0,Y 444.779,Z 674.825,A -85,B 0,C 180,E1 -7359.883,E2 -7359.883} C_VEL
LIN {X 0,Y 443.489,Z 688.388,A -85,B 0,C 180,E1 -7361.737,E2 -7361.737} C_VEL
LIN {X 0,Y 442.379,Z 700.441,A -85,B 0,C 180,E1 -7363.725,E2 -7363.725} C_VEL
LIN {X 0,Y 441.483,Z 711.005,A -85,B 0,C 180,E1 -7365.842,E2 -7365.842} C_VEL
LIN {X 0,Y 440.847,Z 719.619,A -85,B 0,C 180,E1 -7367.957,E2 -7367.957} C_VEL
LIN {X 0,Y 440.381,Z 727.255,A -85,B 0,C 180,E1 -7370.328,E2 -7370.328} C_VEL
LIN {X 0,Y 440.121,Z 733.018,A -85,B 0,C 180,E1 -7372.691,E2 -7372.691} C_VEL
LIN {X 0,Y 439.997,Z 737.235,A -85,B 0,C 180,E1 -7375.177,E2 -7375.177} C_VEL
LIN {X 0,Y 439.954,Z 739.675,A -85,B 0,C 180,E1 -7377.656,E2 -7377.656} C_VEL
LIN {X 0,Y 439.951,Z 740.425,A -85,B 0,C 180,E1 -7380.131,E2 -7380.131} C_VEL
LIN {X 0,Y 439.953,Z 739.489,A -85,B 0,C 180,E1 -7382.606,E2 -7382.606} C_VEL
LIN {X 0,Y 439.993,Z 736.836,A -85,B 0,C 180,E1 -7385.085,E2 -7385.085} C_VEL
LIN {X 0,Y 440.118,Z 732.414,A -85,B 0,C 180,E1 -7387.572,E2 -7387.572} C_VEL
LIN {X 0,Y 440.407,Z 726.08,A -85,B 0,C 180,E1 -7390.068,E2 -7390.068} C_VEL
LIN {X 0,Y 440.892,Z 718.138,A -85,B 0,C 180,E1 -7392.442,E2 -7392.442} C_VEL
LIN {X 0,Y 441.611,Z 708.667,A -85,B 0,C 180,E1 -7394.69,E2 -7394.69} C_VEL
LIN {X 0,Y 442.571,Z 697.708,A -85,B 0,C 180,E1 -7396.809,E2 -7396.809} C_VEL
LIN {X 0,Y 443.755,Z 685.267,A -85,B 0,C 180,E1 -7398.797,E2 -7398.797} C_VEL
LIN {X 0,Y 445.136,Z 671.283,A -85,B 0,C 180,E1 -7400.65,E2 -7400.65} C_VEL
LIN {X 0,Y 446.614,Z 656.284,A -85,B 0,C 180,E1 -7402.301,E2 -7402.301} C_VEL
LIN {X 0,Y 448.114,Z 640.389,A -85,B 0,C 180,E1 -7403.75,E2 -7403.75} C_VEL
LIN {X 0,Y 449.573,Z 623.714,A -85,B 0,C 180,E1 -7404.997,E2 -7404.997} C_VEL
LIN {X 0,Y 450.969,Z 605.565,A -85,B 0,C 180,E1 -7406.083,E2 -7406.083} C_VEL
LIN {X 0,Y 452.193,Z 586.81,A -85,B 0,C 180,E1 -7406.946,E2 -7406.946} C_VEL
LIN {X 0,Y 453.148,Z 567.759,A -85,B 0,C 180,E1 -7407.582,E2 -7407.582} C_VEL
LIN {X 0,Y 453.837,Z 546.607,A -85,B 0,C 180,E1 -7408.037,E2 -7408.037} C_VEL
LIN {X 0,Y 458.256,Z 366.504,A -85,B 0,C 180,E1 -7411.315,E2 -7411.315} C_VEL
LIN {X 0,Y 454.172,Z 340.574,A -85,B 0,C 180,E1 -7412.213,E2 -7412.213} C_VEL
LIN {X 0,Y 455.736,Z 321.368,A -85,B 0,C 180,E1 -7414.072,E2 -7414.072} C_VEL
LIN {X 0,Y 449.365,Z 303.02,A -85,B 0,C 180,E1 -7416.607,E2 -7416.607} C_VEL
LIN {X 0,Y 442.233,Z 284.592,A -85,B 0,C 180,E1 -7419.353,E2 -7419.353} C_VEL
LIN {X 0,Y 441.199,Z 281.714,A -85,B 0,C 180,E1 -7419.851,E2 -7419.851} C_VEL
LIN {X 0,Y 441.193,Z 281.525,A -85,B 0,C 180,E1 -7423.513,E2 -7423.513} C_VEL
LIN {X 0,Y 441.195,Z 281.525,A -85,B 0,C 180,E1 -7427.342,E2 -7427.342} C_VEL
LIN {X 0,Y 441.192,Z 281.529,A -85,B 0,C 180,E1 -7430.388,E2 -7430.388} C_VEL
LIN {X 0,Y 440.226,Z 281.651,A -85,B 0,C 180,E1 -7431.389,E2 -7431.389} C_VEL
LIN {X 0,Y 433.688,Z 282.466,A -85,B 0,C 180,E1 -7434.278,E2 -7434.278} C_VEL
LIN {X 0,Y 433.246,Z 282.517,A -85,B 0,C 180,E1 -7434.941,E2 -7434.941} C_VEL
LIN {X 0,Y 433.246,Z 282.516,A -85,B 0,C 180,E1 -7438.716,E2 -7438.716} C_VEL
LIN {X 0,Y 433.248,Z 282.519,A -85,B 0,C 180,E1 -7442.511,E2 -7442.511} C_VEL
LIN {X 0,Y 433.251,Z 282.513,A -85,B 0,C 180,E1 -7446.323,E2 -7446.323} C_VEL
LIN {X 0,Y 433.259,Z 282.516,A -85,B 0,C 180,E1 -7450.027,E2 -7450.027} C_VEL
LIN {X 0,Y 433.254,Z 282.505,A -85,B 0,C 180,E1 -7453.921,E2 -7453.921} C_VEL
LIN {X 0,Y 433.248,Z 282.789,A -85,B 0,C 180,E1 -7454.66,E2 -7454.66} C_VEL
LIN {X 0,Y 440.653,Z 303.028,A -85,B 0,C 180,E1 -7457.217,E2 -7457.217} C_VEL
LIN {X 0,Y 445.747,Z 318.928,A -85,B 0,C 180,E1 -7459.073,E2 -7459.073} C_VEL
LIN {X 0,Y 444.169,Z 360.129,A -85,B 0,C 180,E1 -7462.692,E2 -7462.692} C_VEL
LIN {X 0,Y 442.449,Z 402.117,A -85,B 0,C 180,E1 -7466.371,E2 -7466.371} C_VEL
LIN {X 0,Y 440.609,Z 445.061,A -85,B 0,C 180,E1 -7470.129,E2 -7470.129} C_VEL
LIN {X 0,Y 439.376,Z 477.348,A -85,B 0,C 180,E1 -7472.927,E2 -7472.927} C_VEL
LIN {X 0,Y 440.893,Z 492.134,A -85,B 0,C 180,E1 -7473.267,E2 -7473.267} C_VEL
LIN {X 0,Y 439.134,Z 620.462,A -85,B 0,C 180,E1 -7475.429,E2 -7475.429} C_VEL
LIN {X 0,Y 438.677,Z 636.459,A -85,B 0,C 180,E1 -7475.939,E2 -7475.939} C_VEL
LIN {X 0,Y 437.958,Z 652.869,A -85,B 0,C 180,E1 -7476.726,E2 -7476.726} C_VEL
LIN {X 0,Y 437.106,Z 667.453,A -85,B 0,C 180,E1 -7477.689,E2 -7477.689} C_VEL
LIN {X 0,Y 436.156,Z 681.295,A -85,B 0,C 180,E1 -7478.867,E2 -7478.867} C_VEL
LIN {X 0,Y 435.218,Z 693.946,A -85,B 0,C 180,E1 -7480.228,E2 -7480.228} C_VEL
LIN {X 0,Y 434.264,Z 706.231,A -85,B 0,C 180,E1 -7481.891,E2 -7481.891} C_VEL
LIN {X 0,Y 433.495,Z 716.267,A -85,B 0,C 180,E1 -7483.605,E2 -7483.605} C_VEL
LIN {X 0,Y 432.856,Z 725.39,A -85,B 0,C 180,E1 -7485.583,E2 -7485.583} C_VEL
LIN {X 0,Y 432.451,Z 732.108,A -85,B 0,C 180,E1 -7487.49,E2 -7487.49} C_VEL
LIN {X 0,Y 432.186,Z 737.739,A -85,B 0,C 180,E1 -7489.677,E2 -7489.677} C_VEL
LIN {X 0,Y 432.068,Z 741.172,A -85,B 0,C 180,E1 -7491.73,E2 -7491.73} C_VEL
LIN {X 0,Y 432.025,Z 743.034,A -85,B 0,C 180,E1 -7493.91,E2 -7493.91} C_VEL
LIN {X 0,Y 432.025,Z 743.18,A -85,B 0,C 180,E1 -7495.937,E2 -7495.937} C_VEL
LIN {X 0,Y 432.067,Z 741.49,A -85,B 0,C 180,E1 -7498.168,E2 -7498.168} C_VEL
LIN {X 0,Y 432.191,Z 738.024,A -85,B 0,C 180,E1 -7500.352,E2 -7500.352} C_VEL
LIN {X 0,Y 432.442,Z 732.785,A -85,B 0,C 180,E1 -7502.442,E2 -7502.442} C_VEL
LIN {X 0,Y 432.872,Z 725.848,A -85,B 0,C 180,E1 -7504.463,E2 -7504.463} C_VEL
LIN {X 0,Y 433.495,Z 717.09,A -85,B 0,C 180,E1 -7506.392,E2 -7506.392} C_VEL
LIN {X 0,Y 434.261,Z 707.32,A -85,B 0,C 180,E1 -7508.099,E2 -7508.099} C_VEL
LIN {X 0,Y 435.168,Z 695.801,A -85,B 0,C 180,E1 -7509.696,E2 -7509.696} C_VEL
LIN {X 0,Y 436.161,Z 682.809,A -85,B 0,C 180,E1 -7511.139,E2 -7511.139} C_VEL
LIN {X 0,Y 437.14,Z 668.595,A -85,B 0,C 180,E1 -7512.371,E2 -7512.371} C_VEL
LIN {X 0,Y 438.03,Z 653.898,A -85,B 0,C 180,E1 -7513.357,E2 -7513.357} C_VEL
LIN {X 0,Y 438.742,Z 637.746,A -85,B 0,C 180,E1 -7514.145,E2 -7514.145} C_VEL
LIN {X 0,Y 439.21,Z 621.585,A -85,B 0,C 180,E1 -7514.676,E2 -7514.676} C_VEL
LIN {X 0,Y 439.971,Z 565.077,A -85,B 0,C 180,E1 -7515.655,E2 -7515.655} C_VEL
LIN {X 0,Y 440.868,Z 488.855,A -85,B 0,C 180,E1 -7516.936,E2 -7516.936} C_VEL
LIN {X 0,Y 439.554,Z 477.444,A -85,B 0,C 180,E1 -7517.234,E2 -7517.234} C_VEL
LIN {X 0,Y 441.159,Z 434.521,A -85,B 0,C 180,E1 -7520.944,E2 -7520.944} C_VEL
LIN {X 0,Y 443.037,Z 389.151,A -85,B 0,C 180,E1 -7524.865,E2 -7524.865} C_VEL
LIN {X 0,Y 444.504,Z 345.174,A -85,B 0,C 180,E1 -7528.618,E2 -7528.618} C_VEL
LIN {X 0,Y 445.246,Z 316.819,A -85,B 0,C 180,E1 -7531.057,E2 -7531.057} C_VEL
LIN {X 0,Y 438.945,Z 297.654,A -85,B 0,C 180,E1 -7533.263,E2 -7533.263} C_VEL
LIN {X 0,Y 433.278,Z 282.866,A -85,B 0,C 180,E1 -7535.125,E2 -7535.125} C_VEL
LIN {X 0,Y 433.223,Z 282.522,A -85,B 0,C 180,E1 -7535.743,E2 -7535.743} C_VEL
LIN {X 0,Y 433.219,Z 282.519,A -85,B 0,C 180,E1 -7539.554,E2 -7539.554} C_VEL
LIN {X 0,Y 433.221,Z 282.523,A -85,B 0,C 180,E1 -7543.37,E2 -7543.37} C_VEL
LIN {X 0,Y 433.239,Z 282.518,A -85,B 0,C 180,E1 -7547.063,E2 -7547.063} C_VEL
LIN {X 0,Y 433.257,Z 282.516,A -85,B 0,C 180,E1 -7550.837,E2 -7550.837} C_VEL
LIN {X 0,Y 433.258,Z 282.52,A -85,B 0,C 180,E1 -7554.57,E2 -7554.57} C_VEL
LIN {X 0,Y 433.25,Z 282.516,A -85,B 0,C 180,E1 -7558.413,E2 -7558.413} C_VEL
LIN {X 0,Y 433.231,Z 282.518,A -85,B 0,C 180,E1 -7562.116,E2 -7562.116} C_VEL
LIN {X 0,Y 433.223,Z 282.52,A -85,B 0,C 180,E1 -7565.908,E2 -7565.908} C_VEL
LIN {X 0,Y 433.225,Z 282.514,A -85,B 0,C 180,E1 -7569.785,E2 -7569.785} C_VEL
LIN {X 0,Y 433.229,Z 282.517,A -85,B 0,C 180,E1 -7573.615,E2 -7573.615} C_VEL
LIN {X 0,Y 433.247,Z 282.516,A -85,B 0,C 180,E1 -7577.32,E2 -7577.32} C_VEL
LIN {X 0,Y 433.262,Z 282.513,A -85,B 0,C 180,E1 -7581.1,E2 -7581.1} C_VEL
LIN {X 0,Y 433.261,Z 282.515,A -85,B 0,C 180,E1 -7584.918,E2 -7584.918} C_VEL
LIN {X 0,Y 433.263,Z 282.518,A -85,B 0,C 180,E1 -7588.729,E2 -7588.729} C_VEL
LIN {X 0,Y 433.242,Z 282.518,A -85,B 0,C 180,E1 -7592.529,E2 -7592.529} C_VEL
LIN {X 0,Y 433.229,Z 282.518,A -85,B 0,C 180,E1 -7596.215,E2 -7596.215} C_VEL
LIN {X 0,Y 433.231,Z 282.518,A -85,B 0,C 180,E1 -7600.083,E2 -7600.083} C_VEL
LIN {X 0,Y 433.24,Z 282.521,A -85,B 0,C 180,E1 -7603.817,E2 -7603.817} C_VEL
LIN {X 0,Y 433.28,Z 282.785,A -85,B 0,C 180,E1 -7606.605,E2 -7606.605} C_VEL
LIN {X 0,Y 442.336,Z 304.575,A -85,B 0,C 180,E1 -7609.819,E2 -7609.819} C_VEL
LIN {X 0,Y 447.798,Z 318.027,A -85,B 0,C 180,E1 -7611.602,E2 -7611.602} C_VEL
LIN {X 0,Y 454.373,Z 330.66,A -85,B 0,C 180,E1 -7612.467,E2 -7612.467} C_VEL
LIN {X 0,Y 456.144,Z 344.815,A -85,B 0,C 180,E1 -7612.924,E2 -7612.924} C_VEL
LIN {X 0,Y 450.988,Z 527.844,A -85,B 0,C 180,E1 -7616.297,E2 -7616.297} C_VEL
LIN {X 0,Y 449.614,Z 578.4,A -85,B 0,C 180,E1 -7617.245,E2 -7617.245} C_VEL
LIN {X 0,Y 448.508,Z 599.317,A -85,B 0,C 180,E1 -7617.859,E2 -7617.859} C_VEL
LIN {X 0,Y 447.058,Z 619.962,A -85,B 0,C 180,E1 -7618.71,E2 -7618.71} C_VEL
LIN {X 0,Y 445.444,Z 639.254,A -85,B 0,C 180,E1 -7619.75,E2 -7619.75} C_VEL
LIN {X 0,Y 443.639,Z 658.179,A -85,B 0,C 180,E1 -7621.018,E2 -7621.018} C_VEL
LIN {X 0,Y 441.751,Z 676.334,A -85,B 0,C 180,E1 -7622.503,E2 -7622.503} C_VEL
LIN {X 0,Y 439.792,Z 694.198,A -85,B 0,C 180,E1 -7624.265,E2 -7624.265} C_VEL
LIN {X 0,Y 437.917,Z 710.869,A -85,B 0,C 180,E1 -7626.237,E2 -7626.237} C_VEL
LIN {X 0,Y 436.365,Z 724.971,A -85,B 0,C 180,E1 -7628.212,E2 -7628.212} C_VEL
LIN {X 0,Y 434.99,Z 738.152,A -85,B 0,C 180,E1 -7630.393,E2 -7630.393} C_VEL
LIN {X 0,Y 433.82,Z 750.534,A -85,B 0,C 180,E1 -7632.844,E2 -7632.844} C_VEL
LIN {X 0,Y 432.96,Z 761.231,A -85,B 0,C 180,E1 -7635.422,E2 -7635.422} C_VEL
LIN {X 0,Y 432.416,Z 769.799,A -85,B 0,C 180,E1 -7637.99,E2 -7637.99} C_VEL
LIN {X 0,Y 432.115,Z 776.509,A -85,B 0,C 180,E1 -7640.546,E2 -7640.546} C_VEL
LIN {X 0,Y 431.987,Z 781.745,A -85,B 0,C 180,E1 -7643.222,E2 -7643.222} C_VEL
LIN {X 0,Y 431.948,Z 785.092,A -85,B 0,C 180,E1 -7645.754,E2 -7645.754} C_VEL
LIN {X 0,Y 431.946,Z 786.854,A -85,B 0,C 180,E1 -7648.277,E2 -7648.277} C_VEL
LIN {X 0,Y 431.953,Z 787.069,A -85,B 0,C 180,E1 -7650.797,E2 -7650.797} C_VEL
LIN {X 0,Y 431.945,Z 785.687,A -85,B 0,C 180,E1 -7653.452,E2 -7653.452} C_VEL
LIN {X 0,Y 431.975,Z 782.803,A -85,B 0,C 180,E1 -7655.98,E2 -7655.98} C_VEL
LIN {X 0,Y 432.075,Z 777.952,A -85,B 0,C 180,E1 -7658.652,E2 -7658.652} C_VEL
LIN {X 0,Y 432.298,Z 771.561,A -85,B 0,C 180,E1 -7661.204,E2 -7661.204} C_VEL
LIN {X 0,Y 432.741,Z 763.295,A -85,B 0,C 180,E1 -7663.769,E2 -7663.769} C_VEL
LIN {X 0,Y 433.418,Z 753.53,A -85,B 0,C 180,E1 -7666.21,E2 -7666.21} C_VEL
LIN {X 0,Y 434.338,Z 742.313,A -85,B 0,C 180,E1 -7668.524,E2 -7668.524} C_VEL
LIN {X 0,Y 435.481,Z 729.664,A -85,B 0,C 180,E1 -7670.708,E2 -7670.708} C_VEL
LIN {X 0,Y 436.89,Z 715.019,A -85,B 0,C 180,E1 -7672.826,E2 -7672.826} C_VEL
LIN {X 0,Y 438.368,Z 699.902,A -85,B 0,C 180,E1 -7674.672,E2 -7674.672} C_VEL
LIN {X 0,Y 439.988,Z 683.393,A -85,B 0,C 180,E1 -7676.378,E2 -7676.378} C_VEL
LIN {X 0,Y 441.659,Z 665.268,A -85,B 0,C 180,E1 -7677.946,E2 -7677.946} C_VEL
LIN {X 0,Y 443.315,Z 646.208,A -85,B 0,C 180,E1 -7679.304,E2 -7679.304} C_VEL
LIN {X 0,Y 444.827,Z 626.726,A -85,B 0,C 180,E1 -7680.43,E2 -7680.43} C_VEL
LIN {X 0,Y 446.19,Z 606.313,A -85,B 0,C 180,E1 -7681.355,E2 -7681.355} C_VEL
LIN {X 0,Y 447.344,Z 585.056,A -85,B 0,C 180,E1 -7682.068,E2 -7682.068} C_VEL
LIN {X 0,Y 448.156,Z 562.417,A -85,B 0,C 180,E1 -7682.577,E2 -7682.577} C_VEL
LIN {X 0,Y 450.521,Z 476.99,A -85,B 0,C 180,E1 -7684.22,E2 -7684.22} C_VEL
LIN {X 0,Y 454.064,Z 394.65,A -85,B 0,C 180,E1 -7686.002,E2 -7686.002} C_VEL
LIN {X 0,Y 456.926,Z 342.616,A -85,B 0,C 180,E1 -7687.247,E2 -7687.247} C_VEL
LIN {X 0,Y 455.948,Z 331.016,A -85,B 0,C 180,E1 -7687.764,E2 -7687.764} C_VEL
LIN {X 0,Y 452.344,Z 323.393,A -85,B 0,C 180,E1 -7688.604,E2 -7688.604} C_VEL
LIN {X 0,Y 450.124,Z 316.137,A -85,B 0,C 180,E1 -7690.105,E2 -7690.105} C_VEL
LIN {X 0,Y 448.031,Z 310.491,A -85,B 0,C 180,E1 -7691.686,E2 -7691.686} C_VEL
LIN {X 0,Y 446.844,Z 307.472,A -85,B 0,C 180,E1 -7692.863,E2 -7692.863} C_VEL
LIN {X 0,Y 445.826,Z 304.501,A -85,B 0,C 180,E1 -7694.767,E2 -7694.767} C_VEL
LIN {X 0,Y 445.598,Z 304.07,A -85,B 0,C 180,E1 -7696.46,E2 -7696.46} C_VEL
LIN {X 0,Y 445.761,Z 305.238,A -85,B 0,C 180,E1 -7697.75,E2 -7697.75} C_VEL
LIN {X 0,Y 446.996,Z 308.181,A -85,B 0,C 180,E1 -7699.558,E2 -7699.558} C_VEL
LIN {X 0,Y 448.407,Z 312.469,A -85,B 0,C 180,E1 -7701.097,E2 -7701.097} C_VEL
LIN {X 0,Y 450.359,Z 318.322,A -85,B 0,C 180,E1 -7702.693,E2 -7702.693} C_VEL
LIN {X 0,Y 452.74,Z 326.881,A -85,B 0,C 180,E1 -7704.492,E2 -7704.492} C_VEL
LIN {X 0,Y 453.286,Z 330.32,A -85,B 0,C 180,E1 -7705.082,E2 -7705.082} C_VEL
LIN {X 0,Y 452.239,Z 337.786,A -85,B 0,C 180,E1 -7705.879,E2 -7705.879} C_VEL
LIN {X 0,Y 454.73,Z 358.347,A -85,B 0,C 180,E1 -7707.041,E2 -7707.041} C_VEL
LIN {X 0,Y 455.701,Z 370.503,A -85,B 0,C 180,E1 -7707.586,E2 -7707.586} C_VEL
LIN {X 0,Y 450.401,Z 454.66,A -85,B 0,C 180,E1 -7709.612,E2 -7709.612} C_VEL
LIN {X 0,Y 446.946,Z 535.528,A -85,B 0,C 180,E1 -7711.397,E2 -7711.397} C_VEL
LIN {X 0,Y 445.747,Z 567.218,A -85,B 0,C 180,E1 -7712.109,E2 -7712.109} C_VEL
LIN {X 0,Y 444.656,Z 587.344,A -85,B 0,C 180,E1 -7712.801,E2 -7712.801} C_VEL
LIN {X 0,Y 443.348,Z 606.589,A -85,B 0,C 180,E1 -7713.708,E2 -7713.708} C_VEL
LIN {X 0,Y 441.885,Z 625.098,A -85,B 0,C 180,E1 -7714.836,E2 -7714.836} C_VEL
LIN {X 0,Y 440.346,Z 642.497,A -85,B 0,C 180,E1 -7716.161,E2 -7716.161} C_VEL
LIN {X 0,Y 438.777,Z 658.936,A -85,B 0,C 180,E1 -7717.696,E2 -7717.696} C_VEL
LIN {X 0,Y 437.236,Z 674.245,A -85,B 0,C 180,E1 -7719.432,E2 -7719.432} C_VEL
LIN {X 0,Y 435.822,Z 688.217,A -85,B 0,C 180,E1 -7721.354,E2 -7721.354} C_VEL
LIN {X 0,Y 434.601,Z 700.641,A -85,B 0,C 180,E1 -7723.425,E2 -7723.425} C_VEL
LIN {X 0,Y 433.639,Z 711.27,A -85,B 0,C 180,E1 -7725.581,E2 -7725.581} C_VEL
LIN {X 0,Y 432.914,Z 720.399,A -85,B 0,C 180,E1 -7727.868,E2 -7727.868} C_VEL
LIN {X 0,Y 432.446,Z 727.626,A -85,B 0,C 180,E1 -7730.149,E2 -7730.149} C_VEL
LIN {X 0,Y 432.157,Z 733.425,A -85,B 0,C 180,E1 -7732.556,E2 -7732.556} C_VEL
LIN {X 0,Y 432.019,Z 737.66,A -85,B 0,C 180,E1 -7735.088,E2 -7735.088} C_VEL
LIN {X 0,Y 431.968,Z 740.113,A -85,B 0,C 180,E1 -7737.613,E2 -7737.613} C_VEL
LIN {X 0,Y 431.962,Z 740.853,A -85,B 0,C 180,E1 -7740.133,E2 -7740.133} C_VEL
LIN {X 0,Y 431.965,Z 739.896,A -85,B 0,C 180,E1 -7742.654,E2 -7742.654} C_VEL
LIN {X 0,Y 432.011,Z 737.223,A -85,B 0,C 180,E1 -7745.179,E2 -7745.179} C_VEL
LIN {X 0,Y 432.149,Z 732.756,A -85,B 0,C 180,E1 -7747.713,E2 -7747.713} C_VEL
LIN {X 0,Y 432.446,Z 726.765,A -85,B 0,C 180,E1 -7750.121,E2 -7750.121} C_VEL
LIN {X 0,Y 432.96,Z 718.88,A -85,B 0,C 180,E1 -7752.538,E2 -7752.538} C_VEL
LIN {X 0,Y 433.719,Z 709.466,A -85,B 0,C 180,E1 -7754.827,E2 -7754.827} C_VEL
LIN {X 0,Y 434.73,Z 698.574,A -85,B 0,C 180,E1 -7756.984,E2 -7756.984} C_VEL
LIN {X 0,Y 435.975,Z 686.215,A -85,B 0,C 180,E1 -7759.006,E2 -7759.006} C_VEL
LIN {X 0,Y 437.425,Z 672.336,A -85,B 0,C 180,E1 -7760.891,E2 -7760.891} C_VEL
LIN {X 0,Y 438.965,Z 657.587,A -85,B 0,C 180,E1 -7762.558,E2 -7762.558} C_VEL
LIN {X 0,Y 440.547,Z 641.772,A -85,B 0,C 180,E1 -7764.042,E2 -7764.042} C_VEL
LIN {X 0,Y 442.133,Z 624.598,A -85,B 0,C 180,E1 -7765.358,E2 -7765.358} C_VEL
LIN {X 0,Y 443.568,Z 607.09,A -85,B 0,C 180,E1 -7766.436,E2 -7766.436} C_VEL
LIN {X 0,Y 444.898,Z 587.883,A -85,B 0,C 180,E1 -7767.348,E2 -7767.348} C_VEL
LIN {X 0,Y 445.932,Z 568.563,A -85,B 0,C 180,E1 -7768.013,E2 -7768.013} C_VEL
LIN {X 0,Y 446.686,Z 547.242,A -85,B 0,C 180,E1 -7768.487,E2 -7768.487} C_VEL
LIN {X 0,Y 451.439,Z 367.771,A -85,B 0,C 180,E1 -7771.827,E2 -7771.827} C_VEL
LIN {X 0,Y 447.208,Z 340.629,A -85,B 0,C 180,E1 -7772.79,E2 -7772.79} C_VEL
LIN {X 0,Y 448.49,Z 324.02,A -85,B 0,C 180,E1 -7774.423,E2 -7774.423} C_VEL
LIN {X 0,Y 442.075,Z 305.546,A -85,B 0,C 180,E1 -7777.022,E2 -7777.022} C_VEL
LIN {X 0,Y 434.556,Z 286.085,A -85,B 0,C 180,E1 -7779.986,E2 -7779.986} C_VEL
LIN {X 0,Y 433.271,Z 282.713,A -85,B 0,C 180,E1 -7780.578,E2 -7780.578} C_VEL
LIN {X 0,Y 433.242,Z 282.512,A -85,B 0,C 180,E1 -7784.37,E2 -7784.37} C_VEL
LIN {X 0,Y 433.246,Z 282.52,A -85,B 0,C 180,E1 -7788.197,E2 -7788.197} C_VEL
LIN {X 0,Y 433.25,Z 282.517,A -85,B 0,C 180,E1 -7791.961,E2 -7791.961} C_VEL
LIN {X 0,Y 433.246,Z 282.517,A -85,B 0,C 180,E1 -7794.941,E2 -7794.941} C_VEL
LIN {X 0,Y 432.246,Z 282.642,A -85,B 0,C 180,E1 -7795.96,E2 -7795.96} C_VEL
LIN {X 0,Y 425.723,Z 283.455,A -85,B 0,C 180,E1 -7798.903,E2 -7798.903} C_VEL
LIN {X 0,Y 425.317,Z 283.497,A -85,B 0,C 180,E1 -7799.578,E2 -7799.578} C_VEL
LIN {X 0,Y 425.297,Z 283.507,A -85,B 0,C 180,E1 -7803.317,E2 -7803.317} C_VEL
LIN {X 0,Y 425.287,Z 283.51,A -85,B 0,C 180,E1 -7807.163,E2 -7807.163} C_VEL
LIN {X 0,Y 425.278,Z 283.509,A -85,B 0,C 180,E1 -7810.934,E2 -7810.934} C_VEL
LIN {X 0,Y 425.351,Z 283.75,A -85,B 0,C 180,E1 -7814.036,E2 -7814.036} C_VEL
LIN {X 0,Y 432.833,Z 303.892,A -85,B 0,C 180,E1 -7816.643,E2 -7816.643} C_VEL
LIN {X 0,Y 438.539,Z 321.631,A -85,B 0,C 180,E1 -7818.758,E2 -7818.758} C_VEL
LIN {X 0,Y 436.845,Z 363.163,A -85,B 0,C 180,E1 -7822.436,E2 -7822.436} C_VEL
LIN {X 0,Y 435.001,Z 404.586,A -85,B 0,C 180,E1 -7826.111,E2 -7826.111} C_VEL
LIN {X 0,Y 433.138,Z 446.443,A -85,B 0,C 180,E1 -7829.8,E2 -7829.8} C_VEL
LIN {X 0,Y 431.886,Z 477.718,A -85,B 0,C 180,E1 -7832.533,E2 -7832.533} C_VEL
LIN {X 0,Y 433.448,Z 492.914,A -85,B 0,C 180,E1 -7832.891,E2 -7832.891} C_VEL
LIN {X 0,Y 431.587,Z 620.801,A -85,B 0,C 180,E1 -7835.082,E2 -7835.082} C_VEL
LIN {X 0,Y 431.105,Z 636.833,A -85,B 0,C 180,E1 -7835.602,E2 -7835.602} C_VEL
LIN {X 0,Y 430.349,Z 653.229,A -85,B 0,C 180,E1 -7836.401,E2 -7836.401} C_VEL
LIN {X 0,Y 429.475,Z 667.498,A -85,B 0,C 180,E1 -7837.355,E2 -7837.355} C_VEL
LIN {X 0,Y 428.443,Z 681.77,A -85,B 0,C 180,E1 -7838.588,E2 -7838.588} C_VEL
LIN {X 0,Y 427.433,Z 694.579,A -85,B 0,C 180,E1 -7839.995,E2 -7839.995} C_VEL
LIN {X 0,Y 426.454,Z 706.448,A -85,B 0,C 180,E1 -7841.631,E2 -7841.631} C_VEL
LIN {X 0,Y 425.661,Z 716.181,A -85,B 0,C 180,E1 -7843.307,E2 -7843.307} C_VEL
LIN {X 0,Y 424.974,Z 725.234,A -85,B 0,C 180,E1 -7845.282,E2 -7845.282} C_VEL
LIN {X 0,Y 424.517,Z 732.222,A -85,B 0,C 180,E1 -7847.262,E2 -7847.262} C_VEL
LIN {X 0,Y 424.22,Z 737.892,A -85,B 0,C 180,E1 -7849.475,E2 -7849.475} C_VEL
LIN {X 0,Y 424.087,Z 741.451,A -85,B 0,C 180,E1 -7851.578,E2 -7851.578} C_VEL
LIN {X 0,Y 424.035,Z 743.381,A -85,B 0,C 180,E1 -7853.808,E2 -7853.808} C_VEL
LIN {X 0,Y 424.036,Z 743.55,A -85,B 0,C 180,E1 -7856.011,E2 -7856.011} C_VEL
LIN {X 0,Y 424.084,Z 741.82,A -85,B 0,C 180,E1 -7858.285,E2 -7858.285} C_VEL
LIN {X 0,Y 424.218,Z 738.441,A -85,B 0,C 180,E1 -7860.445,E2 -7860.445} C_VEL
LIN {X 0,Y 424.504,Z 733.024,A -85,B 0,C 180,E1 -7862.639,E2 -7862.639} C_VEL
LIN {X 0,Y 424.978,Z 726.004,A -85,B 0,C 180,E1 -7864.703,E2 -7864.703} C_VEL
LIN {X 0,Y 425.641,Z 717.38,A -85,B 0,C 180,E1 -7866.629,E2 -7866.629} C_VEL
LIN {X 0,Y 426.485,Z 707.323,A -85,B 0,C 180,E1 -7868.406,E2 -7868.406} C_VEL
LIN {X 0,Y 427.46,Z 695.706,A -85,B 0,C 180,E1 -7870.032,E2 -7870.032} C_VEL
LIN {X 0,Y 428.436,Z 683.67,A -85,B 0,C 180,E1 -7871.39,E2 -7871.39} C_VEL
LIN {X 0,Y 429.46,Z 669.725,A -85,B 0,C 180,E1 -7872.632,E2 -7872.632} C_VEL
LIN {X 0,Y 430.431,Z 654.607,A -85,B 0,C 180,E1 -7873.674,E2 -7873.674} C_VEL
LIN {X 0,Y 431.18,Z 638.651,A -85,B 0,C 180,E1 -7874.472,E2 -7874.472} C_VEL
LIN {X 0,Y 431.689,Z 622.404,A -85,B 0,C 180,E1 -7875.023,E2 -7875.023} C_VEL
LIN {X 0,Y 432.325,Z 578.125,A -85,B 0,C 180,E1 -7875.816,E2 -7875.816} C_VEL
LIN {X 0,Y 433.48,Z 489.716,A -85,B 0,C 180,E1 -7877.329,E2 -7877.329} C_VEL
LIN {X 0,Y 432.105,Z 477.371,A -85,B 0,C 180,E1 -7877.673,E2 -7877.673} C_VEL
LIN {X 0,Y 433.819,Z 434.461,A -85,B 0,C 180,E1 -7881.423,E2 -7881.423} C_VEL
LIN {X 0,Y 435.72,Z 390.732,A -85,B 0,C 180,E1 -7885.233,E2 -7885.233} C_VEL
LIN {X 0,Y 437.267,Z 348.437,A -85,B 0,C 180,E1 -7888.883,E2 -7888.883} C_VEL
LIN {X 0,Y 438.139,Z 319.782,A -85,B 0,C 180,E1 -7891.364,E2 -7891.364} C_VEL
LIN {X 0,Y 432.043,Z 301.18,A -85,B 0,C 180,E1 -7893.544,E2 -7893.544} C_VEL
LIN {X 0,Y 426.068,Z 286.111,A -85,B 0,C 180,E1 -7895.457,E2 -7895.457} C_VEL
LIN {X 0,Y 425.333,Z 283.825,A -85,B 0,C 180,E1 -7895.792,E2 -7895.792} C_VEL
LIN {X 0,Y 425.305,Z 283.504,A -85,B 0,C 180,E1 -7896.883,E2 -7896.883} C_VEL
LIN {X 0,Y 425.319,Z 283.502,A -85,B 0,C 180,E1 -7900.641,E2 -7900.641} C_VEL
LIN {X 0,Y 425.322,Z 283.497,A -85,B 0,C 180,E1 -7904.536,E2 -7904.536} C_VEL
LIN {X 0,Y 425.31,Z 283.513,A -85,B 0,C 180,E1 -7908.335,E2 -7908.335} C_VEL
LIN {X 0,Y 425.299,Z 283.508,A -85,B 0,C 180,E1 -7912.162,E2 -7912.162} C_VEL
LIN {X 0,Y 425.288,Z 283.507,A -85,B 0,C 180,E1 -7915.955,E2 -7915.955} C_VEL
LIN {X 0,Y 425.284,Z 283.508,A -85,B 0,C 180,E1 -7919.73,E2 -7919.73} C_VEL
LIN {X 0,Y 425.288,Z 283.505,A -85,B 0,C 180,E1 -7923.504,E2 -7923.504} C_VEL
LIN {X 0,Y 425.304,Z 283.504,A -85,B 0,C 180,E1 -7927.293,E2 -7927.293} C_VEL
LIN {X 0,Y 425.314,Z 283.505,A -85,B 0,C 180,E1 -7931.114,E2 -7931.114} C_VEL
LIN {X 0,Y 425.325,Z 283.501,A -85,B 0,C 180,E1 -7934.986,E2 -7934.986} C_VEL
LIN {X 0,Y 425.322,Z 283.501,A -85,B 0,C 180,E1 -7938.93,E2 -7938.93} C_VEL
LIN {X 0,Y 425.327,Z 283.505,A -85,B 0,C 180,E1 -7942.857,E2 -7942.857} C_VEL
LIN {X 0,Y 425.314,Z 283.506,A -85,B 0,C 180,E1 -7946.71,E2 -7946.71} C_VEL
LIN {X 0,Y 425.305,Z 283.507,A -85,B 0,C 180,E1 -7950.517,E2 -7950.517} C_VEL
LIN {X 0,Y 425.296,Z 283.506,A -85,B 0,C 180,E1 -7954.349,E2 -7954.349} C_VEL
LIN {X 0,Y 425.293,Z 283.506,A -85,B 0,C 180,E1 -7958.192,E2 -7958.192} C_VEL
LIN {X 0,Y 425.293,Z 283.51,A -85,B 0,C 180,E1 -7962.069,E2 -7962.069} C_VEL
LIN {X 0,Y 425.336,Z 283.755,A -85,B 0,C 180,E1 -7965.816,E2 -7965.816} C_VEL
LIN {X 0,Y 427.659,Z 289.654,A -85,B 0,C 180,E1 -7966.765,E2 -7966.765} C_VEL
LIN {X 0,Y 435.832,Z 308.948,A -85,B 0,C 180,E1 -7969.61,E2 -7969.61} C_VEL
LIN {X 0,Y 439.693,Z 318.355,A -85,B 0,C 180,E1 -7970.869,E2 -7970.869} C_VEL
LIN {X 0,Y 448.026,Z 334.101,A -85,B 0,C 180,E1 -7971.992,E2 -7971.992} C_VEL
LIN {X 0,Y 449.459,Z 346.034,A -85,B 0,C 180,E1 -7972.381,E2 -7972.381} C_VEL
LIN {X 0,Y 443.856,Z 532.639,A -85,B 0,C 180,E1 -7975.888,E2 -7975.888} C_VEL
LIN {X 0,Y 442.508,Z 578.548,A -85,B 0,C 180,E1 -7976.772,E2 -7976.772} C_VEL
LIN {X 0,Y 441.346,Z 599.416,A -85,B 0,C 180,E1 -7977.397,E2 -7977.397} C_VEL
LIN {X 0,Y 439.789,Z 620.497,A -85,B 0,C 180,E1 -7978.284,E2 -7978.284} C_VEL
LIN {X 0,Y 438.006,Z 640.714,A -85,B 0,C 180,E1 -7979.401,E2 -7979.401} C_VEL
LIN {X 0,Y 436.027,Z 660.308,A -85,B 0,C 180,E1 -7980.764,E2 -7980.764} C_VEL
LIN {X 0,Y 433.998,Z 678.619,A -85,B 0,C 180,E1 -7982.323,E2 -7982.323} C_VEL
LIN {X 0,Y 432.12,Z 694.842,A -85,B 0,C 180,E1 -7983.978,E2 -7983.978} C_VEL
LIN {X 0,Y 430.269,Z 710.469,A -85,B 0,C 180,E1 -7985.861,E2 -7985.861} C_VEL
LIN {X 0,Y 428.577,Z 725.034,A -85,B 0,C 180,E1 -7987.94,E2 -7987.94} C_VEL
LIN {X 0,Y 427.131,Z 738.179,A -85,B 0,C 180,E1 -7990.16,E2 -7990.16} C_VEL
LIN {X 0,Y 425.96,Z 749.911,A -85,B 0,C 180,E1 -7992.517,E2 -7992.517} C_VEL
LIN {X 0,Y 425.078,Z 760.127,A -85,B 0,C 180,E1 -7995.006,E2 -7995.006} C_VEL
LIN {X 0,Y 424.495,Z 768.441,A -85,B 0,C 180,E1 -7997.487,E2 -7997.487} C_VEL
LIN {X 0,Y 424.151,Z 775.609,A -85,B 0,C 180,E1 -8000.182,E2 -8000.182} C_VEL
LIN {X 0,Y 423.991,Z 780.871,A -85,B 0,C 180,E1 -8002.822,E2 -8002.822} C_VEL
LIN {X 0,Y 423.954,Z 784.407,A -85,B 0,C 180,E1 -8005.402,E2 -8005.402} C_VEL
LIN {X 0,Y 423.96,Z 786.292,A -85,B 0,C 180,E1 -8007.974,E2 -8007.974} C_VEL
LIN {X 0,Y 423.962,Z 786.661,A -85,B 0,C 180,E1 -8010.677,E2 -8010.677} C_VEL
LIN {X 0,Y 423.954,Z 785.468,A -85,B 0,C 180,E1 -8013.246,E2 -8013.246} C_VEL
LIN {X 0,Y 423.979,Z 782.673,A -85,B 0,C 180,E1 -8015.822,E2 -8015.822} C_VEL
LIN {X 0,Y 424.067,Z 778.23,A -85,B 0,C 180,E1 -8018.407,E2 -8018.407} C_VEL
LIN {X 0,Y 424.278,Z 772.086,A -85,B 0,C 180,E1 -8021.006,E2 -8021.006} C_VEL
LIN {X 0,Y 424.681,Z 764.479,A -85,B 0,C 180,E1 -8023.504,E2 -8023.504} C_VEL
LIN {X 0,Y 425.338,Z 755.162,A -85,B 0,C 180,E1 -8025.965,E2 -8025.965} C_VEL
LIN {X 0,Y 426.241,Z 744.275,A -85,B 0,C 180,E1 -8028.322,E2 -8028.322} C_VEL
LIN {X 0,Y 427.382,Z 732.017,A -85,B 0,C 180,E1 -8030.545,E2 -8030.545} C_VEL
LIN {X 0,Y 428.859,Z 717.422,A -85,B 0,C 180,E1 -8032.77,E2 -8032.77} C_VEL
LIN {X 0,Y 430.461,Z 702.036,A -85,B 0,C 180,E1 -8034.743,E2 -8034.743} C_VEL
LIN {X 0,Y 432.176,Z 685.587,A -85,B 0,C 180,E1 -8036.522,E2 -8036.522} C_VEL
LIN {X 0,Y 433.919,Z 668.028,A -85,B 0,C 180,E1 -8038.115,E2 -8038.115} C_VEL
LIN {X 0,Y 435.735,Z 648.669,A -85,B 0,C 180,E1 -8039.562,E2 -8039.562} C_VEL
LIN {X 0,Y 437.446,Z 628.182,A -85,B 0,C 180,E1 -8040.798,E2 -8040.798} C_VEL
LIN {X 0,Y 438.907,Z 608.019,A -85,B 0,C 180,E1 -8041.752,E2 -8041.752} C_VEL
LIN {X 0,Y 440.238,Z 585.612,A -85,B 0,C 180,E1 -8042.538,E2 -8042.538} C_VEL
LIN {X 0,Y 441.154,Z 562.58,A -85,B 0,C 180,E1 -8043.076,E2 -8043.076} C_VEL
LIN {X 0,Y 443.749,Z 480.887,A -85,B 0,C 180,E1 -8044.716,E2 -8044.716} C_VEL
LIN {X 0,Y 447.564,Z 402.285,A -85,B 0,C 180,E1 -8046.49,E2 -8046.49} C_VEL
LIN {X 0,Y 451.283,Z 344.071,A -85,B 0,C 180,E1 -8047.946,E2 -8047.946} C_VEL
LIN {X 0,Y 450.626,Z 334.976,A -85,B 0,C 180,E1 -8048.365,E2 -8048.365} C_VEL
LIN {X 0,Y 446.314,Z 326.182,A -85,B 0,C 180,E1 -8049.437,E2 -8049.437} C_VEL
LIN {X 0,Y 445.424,Z 324.189,A -85,B 0,C 180,E1 -8049.774,E2 -8049.774} C_VEL
LIN {X 0,Y 443.689,Z 318.701,A -85,B 0,C 180,E1 -8051.178,E2 -8051.178} C_VEL
LIN {X 0,Y 442.253,Z 314.227,A -85,B 0,C 180,E1 -8052.713,E2 -8052.713} C_VEL
LIN {X 0,Y 441.053,Z 311.15,A -85,B 0,C 180,E1 -8054.65,E2 -8054.65} C_VEL
LIN {X 0,Y 440.811,Z 310.485,A -85,B 0,C 180,E1 -8055.866,E2 -8055.866} C_VEL
LIN {X 0,Y 440.882,Z 310.923,A -85,B 0,C 180,E1 -8057.129,E2 -8057.129} C_VEL
LIN {X 0,Y 441.75,Z 313.755,A -85,B 0,C 180,E1 -8059.147,E2 -8059.147} C_VEL
LIN {X 0,Y 443.04,Z 317.992,A -85,B 0,C 180,E1 -8060.809,E2 -8060.809} C_VEL
LIN {X 0,Y 444.853,Z 323.959,A -85,B 0,C 180,E1 -8062.506,E2 -8062.506} C_VEL
LIN {X 0,Y 446.887,Z 332.274,A -85,B 0,C 180,E1 -8064.31,E2 -8064.31} C_VEL
LIN {X 0,Y 447.136,Z 333.991,A -85,B 0,C 180,E1 -8064.609,E2 -8064.609} C_VEL
LIN {X 0,Y 446.755,Z 337.38,A -85,B 0,C 180,E1 -8064.957,E2 -8064.957} C_VEL
LIN {X 0,Y 448.918,Z 357.315,A -85,B 0,C 180,E1 -8066.187,E2 -8066.187} C_VEL
LIN {X 0,Y 449.97,Z 371.91,A -85,B 0,C 180,E1 -8066.896,E2 -8066.896} C_VEL
LIN {X 0,Y 444.104,Z 453.902,A -85,B 0,C 180,E1 -8068.965,E2 -8068.965} C_VEL
LIN {X 0,Y 440.323,Z 530.109,A -85,B 0,C 180,E1 -8070.74,E2 -8070.74} C_VEL
LIN {X 0,Y 438.743,Z 567.556,A -85,B 0,C 180,E1 -8071.61,E2 -8071.61} C_VEL
LIN {X 0,Y 437.528,Z 588.027,A -85,B 0,C 180,E1 -8072.337,E2 -8072.337} C_VEL
LIN {X 0,Y 436.175,Z 606.498,A -85,B 0,C 180,E1 -8073.228,E2 -8073.228} C_VEL
LIN {X 0,Y 434.621,Z 625.027,A -85,B 0,C 180,E1 -8074.374,E2 -8074.374} C_VEL
LIN {X 0,Y 432.97,Z 642.58,A -85,B 0,C 180,E1 -8075.729,E2 -8075.729} C_VEL
LIN {X 0,Y 431.256,Z 659.501,A -85,B 0,C 180,E1 -8077.334,E2 -8077.334} C_VEL
LIN {X 0,Y 429.585,Z 675.07,A -85,B 0,C 180,E1 -8079.139,E2 -8079.139} C_VEL
LIN {X 0,Y 428.106,Z 688.808,A -85,B 0,C 180,E1 -8081.068,E2 -8081.068} C_VEL
LIN {X 0,Y 426.843,Z 700.897,A -85,B 0,C 180,E1 -8083.115,E2 -8083.115} C_VEL
LIN {X 0,Y 425.79,Z 711.738,A -85,B 0,C 180,E1 -8085.35,E2 -8085.35} C_VEL
LIN {X 0,Y 425.022,Z 720.736,A -85,B 0,C 180,E1 -8087.639,E2 -8087.639} C_VEL
LIN {X 0,Y 424.515,Z 728.003,A -85,B 0,C 180,E1 -8089.963,E2 -8089.963} C_VEL
LIN {X 0,Y 424.193,Z 733.833,A -85,B 0,C 180,E1 -8092.415,E2 -8092.415} C_VEL
LIN {X 0,Y 424.04,Z 738.089,A -85,B 0,C 180,E1 -8094.995,E2 -8094.995} C_VEL
LIN {X 0,Y 423.981,Z 740.549,A -85,B 0,C 180,E1 -8097.568,E2 -8097.568} C_VEL
LIN {X 0,Y 423.974,Z 741.282,A -85,B 0,C 180,E1 -8100.136,E2 -8100.136} C_VEL
LIN {X 0,Y 423.978,Z 740.303,A -85,B 0,C 180,E1 -8102.704,E2 -8102.704} C_VEL
LIN {X 0,Y 424.03,Z 737.598,A -85,B 0,C 180,E1 -8105.277,E2 -8105.277} C_VEL
LIN {X 0,Y 424.181,Z 733.087,A -85,B 0,C 180,E1 -8107.858,E2 -8107.858} C_VEL
LIN {X 0,Y 424.504,Z 727.048,A -85,B 0,C 180,E1 -8110.312,E2 -8110.312} C_VEL
LIN {X 0,Y 425.064,Z 719.102,A -85,B 0,C 180,E1 -8112.775,E2 -8112.775} C_VEL
LIN {X 0,Y 425.885,Z 709.625,A -85,B 0,C 180,E1 -8115.106,E2 -8115.106} C_VEL
LIN {X 0,Y 426.969,Z 698.661,A -85,B 0,C 180,E1 -8117.302,E2 -8117.302} C_VEL
LIN {X 0,Y 428.299,Z 686.217,A -85,B 0,C 180,E1 -8119.36,E2 -8119.36} C_VEL
LIN {X 0,Y 429.837,Z 672.239,A -85,B 0,C 180,E1 -8121.278,E2 -8121.278} C_VEL
LIN {X 0,Y 431.475,Z 657.269,A -85,B 0,C 180,E1 -8122.984,E2 -8122.984} C_VEL
LIN {X 0,Y 433.135,Z 641.442,A -85,B 0,C 180,E1 -8124.48,E2 -8124.48} C_VEL
LIN {X 0,Y 434.813,Z 624.151,A -85,B 0,C 180,E1 -8125.815,E2 -8125.815} C_VEL
LIN {X 0,Y 436.322,Z 606.476,A -85,B 0,C 180,E1 -8126.91,E2 -8126.91} C_VEL
LIN {X 0,Y 437.7,Z 587.49,A -85,B 0,C 180,E1 -8127.818,E2 -8127.818} C_VEL
LIN {X 0,Y 438.784,Z 568.171,A -85,B 0,C 180,E1 -8128.488,E2 -8128.488} C_VEL
LIN {X 0,Y 439.595,Z 546.054,A -85,B 0,C 180,E1 -8128.983,E2 -8128.983} C_VEL
LIN {X 0,Y 444.663,Z 368.932,A -85,B 0,C 180,E1 -8132.363,E2 -8132.363} C_VEL
LIN {X 0,Y 440.269,Z 340.137,A -85,B 0,C 180,E1 -8133.417,E2 -8133.417} C_VEL
LIN {X 0,Y 441.449,Z 327.276,A -85,B 0,C 180,E1 -8134.695,E2 -8134.695} C_VEL
LIN {X 0,Y 434.932,Z 308.602,A -85,B 0,C 180,E1 -8137.367,E2 -8137.367} C_VEL
LIN {X 0,Y 427.944,Z 290.418,A -85,B 0,C 180,E1 -8140.18,E2 -8140.18} C_VEL
LIN {X 0,Y 425.351,Z 283.703,A -85,B 0,C 180,E1 -8141.308,E2 -8141.308} C_VEL
LIN {X 0,Y 425.319,Z 283.506,A -85,B 0,C 180,E1 -8145.149,E2 -8145.149} C_VEL
LIN {X 0,Y 425.316,Z 283.507,A -85,B 0,C 180,E1 -8149.012,E2 -8149.012} C_VEL
LIN {X 0,Y 425.314,Z 283.508,A -85,B 0,C 180,E1 -8152.84,E2 -8152.84} C_VEL
LIN {X 0,Y 425.314,Z 283.507,A -85,B 0,C 180,E1 -8156.625,E2 -8156.625} C_VEL
LIN {X 0,Y 425.317,Z 283.497,A -85,B 0,C 180,E1 -8159.578,E2 -8159.578} C_VEL
LIN {X 0,Y 424.374,Z 283.608,A -85,B 0,C 180,E1 -8160.616,E2 -8160.616} C_VEL
LIN {X 0,Y 417.836,Z 284.436,A -85,B 0,C 180,E1 -8163.614,E2 -8163.614} C_VEL
LIN {X 0,Y 417.374,Z 284.482,A -85,B 0,C 180,E1 -8164.302,E2 -8164.302} C_VEL
LIN {X 0,Y 417.379,Z 284.483,A -85,B 0,C 180,E1 -8168.202,E2 -8168.202} C_VEL
LIN {X 0,Y 417.376,Z 284.484,A -85,B 0,C 180,E1 -8172,E2 -8172} C_VEL
LIN {X 0,Y 417.378,Z 284.754,A -85,B 0,C 180,E1 -8173.383,E2 -8173.383} C_VEL
LIN {X 0,Y 425.129,Z 305.321,A -85,B 0,C 180,E1 -8176.118,E2 -8176.118} C_VEL
LIN {X 0,Y 431.201,Z 323.769,A -85,B 0,C 180,E1 -8178.36,E2 -8178.36} C_VEL
LIN {X 0,Y 430.107,Z 353.014,A -85,B 0,C 180,E1 -8180.997,E2 -8180.997} C_VEL
LIN {X 0,Y 428.203,Z 394.572,A -85,B 0,C 180,E1 -8184.707,E2 -8184.707} C_VEL
LIN {X 0,Y 426.075,Z 438.721,A -85,B 0,C 180,E1 -8188.654,E2 -8188.654} C_VEL
LIN {X 0,Y 424.417,Z 478.081,A -85,B 0,C 180,E1 -8192.125,E2 -8192.125} C_VEL
LIN {X 0,Y 426.023,Z 493.695,A -85,B 0,C 180,E1 -8192.502,E2 -8192.502} C_VEL
LIN {X 0,Y 424.056,Z 621.138,A -85,B 0,C 180,E1 -8194.724,E2 -8194.724} C_VEL
LIN {X 0,Y 423.552,Z 637.168,A -85,B 0,C 180,E1 -8195.251,E2 -8195.251} C_VEL
LIN {X 0,Y 422.779,Z 653.135,A -85,B 0,C 180,E1 -8196.039,E2 -8196.039} C_VEL
LIN {X 0,Y 421.859,Z 667.544,A -85,B 0,C 180,E1 -8197.01,E2 -8197.01} C_VEL
LIN {X 0,Y 420.769,Z 681.882,A -85,B 0,C 180,E1 -8198.264,E2 -8198.264} C_VEL
LIN {X 0,Y 419.719,Z 694.525,A -85,B 0,C 180,E1 -8199.667,E2 -8199.667} C_VEL
LIN {X 0,Y 418.693,Z 706.205,A -85,B 0,C 180,E1 -8201.291,E2 -8201.291} C_VEL
LIN {X 0,Y 417.798,Z 716.532,A -85,B 0,C 180,E1 -8203.087,E2 -8203.087} C_VEL
LIN {X 0,Y 417.048,Z 725.79,A -85,B 0,C 180,E1 -8205.147,E2 -8205.147} C_VEL
LIN {X 0,Y 416.556,Z 732.803,A -85,B 0,C 180,E1 -8207.19,E2 -8207.19} C_VEL
LIN {X 0,Y 416.249,Z 738.236,A -85,B 0,C 180,E1 -8209.357,E2 -8209.357} C_VEL
LIN {X 0,Y 416.1,Z 741.901,A -85,B 0,C 180,E1 -8211.574,E2 -8211.574} C_VEL
LIN {X 0,Y 416.044,Z 743.855,A -85,B 0,C 180,E1 -8213.961,E2 -8213.961} C_VEL
LIN {X 0,Y 416.046,Z 743.917,A -85,B 0,C 180,E1 -8216.089,E2 -8216.089} C_VEL
LIN {X 0,Y 416.104,Z 742.138,A -85,B 0,C 180,E1 -8218.421,E2 -8218.421} C_VEL
LIN {X 0,Y 416.254,Z 738.717,A -85,B 0,C 180,E1 -8220.611,E2 -8220.611} C_VEL
LIN {X 0,Y 416.571,Z 733.245,A -85,B 0,C 180,E1 -8222.851,E2 -8222.851} C_VEL
LIN {X 0,Y 417.081,Z 726.26,A -85,B 0,C 180,E1 -8224.927,E2 -8224.927} C_VEL
LIN {X 0,Y 417.824,Z 717.355,A -85,B 0,C 180,E1 -8226.939,E2 -8226.939} C_VEL
LIN {X 0,Y 418.721,Z 707.313,A -85,B 0,C 180,E1 -8228.726,E2 -8228.726} C_VEL
LIN {X 0,Y 419.836,Z 694.926,A -85,B 0,C 180,E1 -8230.468,E2 -8230.468} C_VEL
LIN {X 0,Y 420.905,Z 682.328,A -85,B 0,C 180,E1 -8231.873,E2 -8231.873} C_VEL
LIN {X 0,Y 422.007,Z 667.978,A -85,B 0,C 180,E1 -8233.134,E2 -8233.134} C_VEL
LIN {X 0,Y 422.954,Z 653.486,A -85,B 0,C 180,E1 -8234.11,E2 -8234.11} C_VEL
LIN {X 0,Y 423.753,Z 636.992,A -85,B 0,C 180,E1 -8234.922,E2 -8234.922} C_VEL
LIN {X 0,Y 424.229,Z 620.962,A -85,B 0,C 180,E1 -8235.438,E2 -8235.438} C_VEL
LIN {X 0,Y 426.104,Z 490.472,A -85,B 0,C 180,E1 -8237.739,E2 -8237.739} C_VEL
LIN {X 0,Y 424.681,Z 478.164,A -85,B 0,C 180,E1 -8238.069,E2 -8238.069} C_VEL
LIN {X 0,Y 426.483,Z 435.275,A -85,B 0,C 180,E1 -8241.847,E2 -8241.847} C_VEL
LIN {X 0,Y 428.431,Z 392.366,A -85,B 0,C 180,E1 -8245.613,E2 -8245.613} C_VEL
LIN {X 0,Y 430.038,Z 351.813,A -85,B 0,C 180,E1 -8249.15,E2 -8249.15} C_VEL
LIN {X 0,Y 430.942,Z 322.307,A -85,B 0,C 180,E1 -8251.75,E2 -8251.75} C_VEL
LIN {X 0,Y 424.84,Z 303.788,A -85,B 0,C 180,E1 -8253.964,E2 -8253.964} C_VEL
LIN {X 0,Y 418.52,Z 287.76,A -85,B 0,C 180,E1 -8256.037,E2 -8256.037} C_VEL
LIN {X 0,Y 417.417,Z 284.724,A -85,B 0,C 180,E1 -8256.502,E2 -8256.502} C_VEL
LIN {X 0,Y 417.371,Z 284.498,A -85,B 0,C 180,E1 -8260.258,E2 -8260.258} C_VEL
LIN {X 0,Y 417.353,Z 284.492,A -85,B 0,C 180,E1 -8264.007,E2 -8264.007} C_VEL
LIN {X 0,Y 417.345,Z 284.499,A -85,B 0,C 180,E1 -8267.804,E2 -8267.804} C_VEL
LIN {X 0,Y 417.344,Z 284.496,A -85,B 0,C 180,E1 -8271.655,E2 -8271.655} C_VEL
LIN {X 0,Y 417.348,Z 284.496,A -85,B 0,C 180,E1 -8275.465,E2 -8275.465} C_VEL
LIN {X 0,Y 417.356,Z 284.496,A -85,B 0,C 180,E1 -8279.313,E2 -8279.313} C_VEL
LIN {X 0,Y 417.365,Z 284.493,A -85,B 0,C 180,E1 -8283.158,E2 -8283.158} C_VEL
LIN {X 0,Y 417.386,Z 284.49,A -85,B 0,C 180,E1 -8287.017,E2 -8287.017} C_VEL
LIN {X 0,Y 417.381,Z 284.495,A -85,B 0,C 180,E1 -8290.908,E2 -8290.908} C_VEL
LIN {X 0,Y 417.386,Z 284.491,A -85,B 0,C 180,E1 -8294.851,E2 -8294.851} C_VEL
LIN {X 0,Y 417.379,Z 284.491,A -85,B 0,C 180,E1 -8298.723,E2 -8298.723} C_VEL
LIN {X 0,Y 417.37,Z 284.492,A -85,B 0,C 180,E1 -8302.538,E2 -8302.538} C_VEL
LIN {X 0,Y 417.359,Z 284.499,A -85,B 0,C 180,E1 -8306.37,E2 -8306.37} C_VEL
LIN {X 0,Y 417.354,Z 284.494,A -85,B 0,C 180,E1 -8310.139,E2 -8310.139} C_VEL
LIN {X 0,Y 417.353,Z 284.495,A -85,B 0,C 180,E1 -8314.016,E2 -8314.016} C_VEL
LIN {X 0,Y 417.359,Z 284.494,A -85,B 0,C 180,E1 -8317.828,E2 -8317.828} C_VEL
LIN {X 0,Y 417.37,Z 284.495,A -85,B 0,C 180,E1 -8321.635,E2 -8321.635} C_VEL
LIN {X 0,Y 417.412,Z 284.728,A -85,B 0,C 180,E1 -8325.015,E2 -8325.015} C_VEL
LIN {X 0,Y 420.168,Z 291.543,A -85,B 0,C 180,E1 -8326.14,E2 -8326.14} C_VEL
LIN {X 0,Y 429.114,Z 312.779,A -85,B 0,C 180,E1 -8329.326,E2 -8329.326} C_VEL
LIN {X 0,Y 431.606,Z 318.766,A -85,B 0,C 180,E1 -8330.118,E2 -8330.118} C_VEL
LIN {X 0,Y 441.707,Z 337.509,A -85,B 0,C 180,E1 -8331.501,E2 -8331.501} C_VEL
LIN {X 0,Y 442.806,Z 347.412,A -85,B 0,C 180,E1 -8331.825,E2 -8331.825} C_VEL
LIN {X 0,Y 436.724,Z 537.254,A -85,B 0,C 180,E1 -8335.469,E2 -8335.469} C_VEL
LIN {X 0,Y 435.415,Z 578.599,A -85,B 0,C 180,E1 -8336.287,E2 -8336.287} C_VEL
LIN {X 0,Y 434.193,Z 599.455,A -85,B 0,C 180,E1 -8336.925,E2 -8336.925} C_VEL
LIN {X 0,Y 432.594,Z 620.027,A -85,B 0,C 180,E1 -8337.802,E2 -8337.802} C_VEL
LIN {X 0,Y 430.742,Z 640.166,A -85,B 0,C 180,E1 -8338.93,E2 -8338.93} C_VEL
LIN {X 0,Y 428.785,Z 658.638,A -85,B 0,C 180,E1 -8340.221,E2 -8340.221} C_VEL
LIN {X 0,Y 426.722,Z 676.673,A -85,B 0,C 180,E1 -8341.753,E2 -8341.753} C_VEL
LIN {X 0,Y 424.692,Z 693.464,A -85,B 0,C 180,E1 -8343.462,E2 -8343.462} C_VEL
LIN {X 0,Y 422.633,Z 709.984,A -85,B 0,C 180,E1 -8345.47,E2 -8345.47} C_VEL
LIN {X 0,Y 420.895,Z 724.267,A -85,B 0,C 180,E1 -8347.531,E2 -8347.531} C_VEL
LIN {X 0,Y 419.364,Z 737.445,A -85,B 0,C 180,E1 -8349.777,E2 -8349.777} C_VEL
LIN {X 0,Y 418.11,Z 749.237,A -85,B 0,C 180,E1 -8352.178,E2 -8352.178} C_VEL
LIN {X 0,Y 417.166,Z 759.532,A -85,B 0,C 180,E1 -8354.715,E2 -8354.715} C_VEL
LIN {X 0,Y 416.539,Z 767.912,A -85,B 0,C 180,E1 -8357.244,E2 -8357.244} C_VEL
LIN {X 0,Y 416.163,Z 775.241,A -85,B 0,C 180,E1 -8360.04,E2 -8360.04} C_VEL
LIN {X 0,Y 415.997,Z 780.424,A -85,B 0,C 180,E1 -8362.683,E2 -8362.683} C_VEL
LIN {X 0,Y 415.961,Z 783.972,A -85,B 0,C 180,E1 -8365.314,E2 -8365.314} C_VEL
LIN {X 0,Y 415.97,Z 785.865,A -85,B 0,C 180,E1 -8367.935,E2 -8367.935} C_VEL
LIN {X 0,Y 415.974,Z 786.226,A -85,B 0,C 180,E1 -8370.69,E2 -8370.69} C_VEL
LIN {X 0,Y 415.965,Z 785.009,A -85,B 0,C 180,E1 -8373.309,E2 -8373.309} C_VEL
LIN {X 0,Y 415.988,Z 782.19,A -85,B 0,C 180,E1 -8375.934,E2 -8375.934} C_VEL
LIN {X 0,Y 416.077,Z 777.698,A -85,B 0,C 180,E1 -8378.57,E2 -8378.57} C_VEL
LIN {X 0,Y 416.298,Z 771.492,A -85,B 0,C 180,E1 -8381.219,E2 -8381.219} C_VEL
LIN {X 0,Y 416.729,Z 763.9,A -85,B 0,C 180,E1 -8383.742,E2 -8383.742} C_VEL
LIN {X 0,Y 417.438,Z 754.436,A -85,B 0,C 180,E1 -8386.276,E2 -8386.276} C_VEL
LIN {X 0,Y 418.479,Z 742.779,A -85,B 0,C 180,E1 -8388.819,E2 -8388.819} C_VEL
LIN {X 0,Y 419.723,Z 730.288,A -85,B 0,C 180,E1 -8391.084,E2 -8391.084} C_VEL
LIN {X 0,Y 421.277,Z 715.819,A -85,B 0,C 180,E1 -8393.292,E2 -8393.292} C_VEL
LIN {X 0,Y 423.02,Z 699.925,A -85,B 0,C 180,E1 -8395.33,E2 -8395.33} C_VEL
LIN {X 0,Y 424.947,Z 682.47,A -85,B 0,C 180,E1 -8397.203,E2 -8397.203} C_VEL
LIN {X 0,Y 426.872,Z 663.986,A -85,B 0,C 180,E1 -8398.851,E2 -8398.851} C_VEL
LIN {X 0,Y 428.718,Z 644.913,A -85,B 0,C 180,E1 -8400.25,E2 -8400.25} C_VEL
LIN {X 0,Y 430.474,Z 625.001,A -85,B 0,C 180,E1 -8401.43,E2 -8401.43} C_VEL
LIN {X 0,Y 432.01,Z 604.551,A -85,B 0,C 180,E1 -8402.383,E2 -8402.383} C_VEL
LIN {X 0,Y 433.366,Z 583.279,A -85,B 0,C 180,E1 -8403.114,E2 -8403.114} C_VEL
LIN {X 0,Y 434.335,Z 560.012,A -85,B 0,C 180,E1 -8403.66,E2 -8403.66} C_VEL
LIN {X 0,Y 437.202,Z 482.276,A -85,B 0,C 180,E1 -8405.297,E2 -8405.297} C_VEL
LIN {X 0,Y 441.361,Z 407.179,A -85,B 0,C 180,E1 -8407.072,E2 -8407.072} C_VEL
LIN {X 0,Y 445.911,Z 345.782,A -85,B 0,C 180,E1 -8408.675,E2 -8408.675} C_VEL
LIN {X 0,Y 445.566,Z 338.925,A -85,B 0,C 180,E1 -8409.015,E2 -8409.015} C_VEL
LIN {X 0,Y 441.709,Z 330.881,A -85,B 0,C 180,E1 -8410.085,E2 -8410.085} C_VEL
LIN {X 0,Y 439.019,Z 325.909,A -85,B 0,C 180,E1 -8410.99,E2 -8410.99} C_VEL
LIN {X 0,Y 437.703,Z 322.033,A -85,B 0,C 180,E1 -8412.259,E2 -8412.259} C_VEL
LIN {X 0,Y 436.917,Z 319.704,A -85,B 0,C 180,E1 -8413.305,E2 -8413.305} C_VEL
LIN {X 0,Y 436.257,Z 317.093,A -85,B 0,C 180,E1 -8415.283,E2 -8415.283} C_VEL
LIN {X 0,Y 436.162,Z 317.206,A -85,B 0,C 180,E1 -8416.911,E2 -8416.911} C_VEL
LIN {X 0,Y 436.83,Z 320.025,A -85,B 0,C 180,E1 -8419.056,E2 -8419.056} C_VEL
LIN {X 0,Y 437.947,Z 324.346,A -85,B 0,C 180,E1 -8420.773,E2 -8420.773} C_VEL
LIN {X 0,Y 439.622,Z 330.524,A -85,B 0,C 180,E1 -8422.539,E2 -8422.539} C_VEL
LIN {X 0,Y 440.842,Z 335.919,A -85,B 0,C 180,E1 -8423.737,E2 -8423.737} C_VEL
LIN {X 0,Y 441.837,Z 339.013,A -85,B 0,C 180,E1 -8424.119,E2 -8424.119} C_VEL
LIN {X 0,Y 443.51,Z 357.592,A -85,B 0,C 180,E1 -8425.346,E2 -8425.346} C_VEL
LIN {X 0,Y 444.469,Z 373.275,A -85,B 0,C 180,E1 -8426.168,E2 -8426.168} C_VEL
LIN {X 0,Y 438.012,Z 452.967,A -85,B 0,C 180,E1 -8428.273,E2 -8428.273} C_VEL
LIN {X 0,Y 433.8,Z 526.459,A -85,B 0,C 180,E1 -8430.078,E2 -8430.078} C_VEL
LIN {X 0,Y 431.85,Z 567.574,A -85,B 0,C 180,E1 -8431.072,E2 -8431.072} C_VEL
LIN {X 0,Y 430.518,Z 588.238,A -85,B 0,C 180,E1 -8431.824,E2 -8431.824} C_VEL
LIN {X 0,Y 429.047,Z 606.93,A -85,B 0,C 180,E1 -8432.747,E2 -8432.747} C_VEL
LIN {X 0,Y 427.395,Z 625.318,A -85,B 0,C 180,E1 -8433.909,E2 -8433.909} C_VEL
LIN {X 0,Y 425.637,Z 642.814,A -85,B 0,C 180,E1 -8435.283,E2 -8435.283} C_VEL
LIN {X 0,Y 423.921,Z 658.661,A -85,B 0,C 180,E1 -8436.804,E2 -8436.804} C_VEL
LIN {X 0,Y 422.223,Z 673.664,A -85,B 0,C 180,E1 -8438.539,E2 -8438.539} C_VEL
LIN {X 0,Y 420.671,Z 687.19,A -85,B 0,C 180,E1 -8440.42,E2 -8440.42} C_VEL
LIN {X 0,Y 419.25,Z 699.883,A -85,B 0,C 180,E1 -8442.547,E2 -8442.547} C_VEL
LIN {X 0,Y 418.111,Z 710.679,A -85,B 0,C 180,E1 -8444.749,E2 -8444.749} C_VEL
LIN {X 0,Y 417.224,Z 720.135,A -85,B 0,C 180,E1 -8447.123,E2 -8447.123} C_VEL
LIN {X 0,Y 416.607,Z 728.023,A -85,B 0,C 180,E1 -8449.631,E2 -8449.631} C_VEL
LIN {X 0,Y 416.233,Z 734.25,A -85,B 0,C 180,E1 -8452.27,E2 -8452.27} C_VEL
LIN {X 0,Y 416.062,Z 738.522,A -85,B 0,C 180,E1 -8454.899,E2 -8454.899} C_VEL
LIN {X 0,Y 415.995,Z 740.986,A -85,B 0,C 180,E1 -8457.521,E2 -8457.521} C_VEL
LIN {X 0,Y 415.986,Z 741.71,A -85,B 0,C 180,E1 -8460.138,E2 -8460.138} C_VEL
LIN {X 0,Y 415.991,Z 740.711,A -85,B 0,C 180,E1 -8462.756,E2 -8462.756} C_VEL
LIN {X 0,Y 416.048,Z 737.973,A -85,B 0,C 180,E1 -8465.379,E2 -8465.379} C_VEL
LIN {X 0,Y 416.215,Z 733.417,A -85,B 0,C 180,E1 -8468.01,E2 -8468.01} C_VEL
LIN {X 0,Y 416.566,Z 727.326,A -85,B 0,C 180,E1 -8470.511,E2 -8470.511} C_VEL
LIN {X 0,Y 417.173,Z 719.314,A -85,B 0,C 180,E1 -8473.021,E2 -8473.021} C_VEL
LIN {X 0,Y 418.06,Z 709.762,A -85,B 0,C 180,E1 -8475.396,E2 -8475.396} C_VEL
LIN {X 0,Y 419.218,Z 698.715,A -85,B 0,C 180,E1 -8477.633,E2 -8477.633} C_VEL
LIN {X 0,Y 420.635,Z 686.186,A -85,B 0,C 180,E1 -8479.727,E2 -8479.727} C_VEL
LIN {X 0,Y 422.266,Z 672.107,A -85,B 0,C 180,E1 -8481.678,E2 -8481.678} C_VEL
LIN {X 0,Y 424.004,Z 656.944,A -85,B 0,C 180,E1 -8483.42,E2 -8483.42} C_VEL
LIN {X 0,Y 425.752,Z 640.958,A -85,B 0,C 180,E1 -8484.94,E2 -8484.94} C_VEL
LIN {X 0,Y 427.445,Z 624.321,A -85,B 0,C 180,E1 -8486.239,E2 -8486.239} C_VEL
LIN {X 0,Y 429.05,Z 606.308,A -85,B 0,C 180,E1 -8487.368,E2 -8487.368} C_VEL
LIN {X 0,Y 430.482,Z 587.36,A -85,B 0,C 180,E1 -8488.283,E2 -8488.283} C_VEL
LIN {X 0,Y 431.624,Z 568.015,A -85,B 0,C 180,E1 -8488.962,E2 -8488.962} C_VEL
LIN {X 0,Y 432.473,Z 545.888,A -85,B 0,C 180,E1 -8489.466,E2 -8489.466} C_VEL
LIN {X 0,Y 437.927,Z 370.277,A -85,B 0,C 180,E1 -8492.903,E2 -8492.903} C_VEL
LIN {X 0,Y 433.368,Z 339.946,A -85,B 0,C 180,E1 -8494.038,E2 -8494.038} C_VEL
LIN {X 0,Y 434.241,Z 329.996,A -85,B 0,C 180,E1 -8495.047,E2 -8495.047} C_VEL
LIN {X 0,Y 428.031,Z 312.209,A -85,B 0,C 180,E1 -8497.636,E2 -8497.636} C_VEL
LIN {X 0,Y 420.921,Z 293.897,A -85,B 0,C 180,E1 -8500.523,E2 -8500.523} C_VEL
LIN {X 0,Y 417.386,Z 284.693,A -85,B 0,C 180,E1 -8502.083,E2 -8502.083} C_VEL
LIN {X 0,Y 417.37,Z 284.496,A -85,B 0,C 180,E1 -8505.802,E2 -8505.802} C_VEL
LIN {X 0,Y 417.38,Z 284.495,A -85,B 0,C 180,E1 -8509.698,E2 -8509.698} C_VEL
LIN {X 0,Y 417.378,Z 284.492,A -85,B 0,C 180,E1 -8513.603,E2 -8513.603} C_VEL
LIN {X 0,Y 417.377,Z 284.492,A -85,B 0,C 180,E1 -8517.546,E2 -8517.546} C_VEL
LIN {X 0,Y 417.364,Z 284.482,A -85,B 0,C 180,E1 -8521.37,E2 -8521.37} C_VEL
LIN {X 0,Y 417.374,Z 284.482,A -85,B 0,C 180,E1 -8524.302,E2 -8524.302} C_VEL
LIN {X 0,Y 416.355,Z 284.611,A -85,B 0,C 180,E1 -8525.36,E2 -8525.36} C_VEL
LIN {X 0,Y 409.833,Z 285.422,A -85,B 0,C 180,E1 -8528.416,E2 -8528.416} C_VEL
LIN {X 0,Y 409.404,Z 285.475,A -85,B 0,C 180,E1 -8529.117,E2 -8529.117} C_VEL
LIN {X 0,Y 409.424,Z 285.654,A -85,B 0,C 180,E1 -8532.665,E2 -8532.665} C_VEL
LIN {X 0,Y 409.945,Z 287.565,A -85,B 0,C 180,E1 -8532.98,E2 -8532.98} C_VEL
LIN {X 0,Y 416.426,Z 303.82,A -85,B 0,C 180,E1 -8535.183,E2 -8535.183} C_VEL
LIN {X 0,Y 423.283,Z 324.023,A -85,B 0,C 180,E1 -8537.724,E2 -8537.724} C_VEL
LIN {X 0,Y 424.155,Z 327.905,A -85,B 0,C 180,E1 -8538.164,E2 -8538.164} C_VEL
LIN {X 0,Y 422.202,Z 369.171,A -85,B 0,C 180,E1 -8541.898,E2 -8541.898} C_VEL
LIN {X 0,Y 420.196,Z 409.88,A -85,B 0,C 180,E1 -8545.563,E2 -8545.563} C_VEL
LIN {X 0,Y 418.12,Z 452.276,A -85,B 0,C 180,E1 -8549.382,E2 -8549.382} C_VEL
LIN {X 0,Y 416.97,Z 478.502,A -85,B 0,C 180,E1 -8551.705,E2 -8551.705} C_VEL
LIN {X 0,Y 418.618,Z 494.474,A -85,B 0,C 180,E1 -8552.099,E2 -8552.099} C_VEL
LIN {X 0,Y 416.535,Z 621.551,A -85,B 0,C 180,E1 -8554.356,E2 -8554.356} C_VEL
LIN {X 0,Y 416.005,Z 637.569,A -85,B 0,C 180,E1 -8554.893,E2 -8554.893} C_VEL
LIN {X 0,Y 415.223,Z 653.003,A -85,B 0,C 180,E1 -8555.664,E2 -8555.664} C_VEL
LIN {X 0,Y 414.257,Z 667.567,A -85,B 0,C 180,E1 -8556.651,E2 -8556.651} C_VEL
LIN {X 0,Y 413.107,Z 681.979,A -85,B 0,C 180,E1 -8557.928,E2 -8557.928} C_VEL
LIN {X 0,Y 411.997,Z 694.7,A -85,B 0,C 180,E1 -8559.356,E2 -8559.356} C_VEL
LIN {X 0,Y 410.863,Z 706.887,A -85,B 0,C 180,E1 -8561.082,E2 -8561.082} C_VEL
LIN {X 0,Y 409.96,Z 716.704,A -85,B 0,C 180,E1 -8562.821,E2 -8562.821} C_VEL
LIN {X 0,Y 409.167,Z 725.785,A -85,B 0,C 180,E1 -8564.866,E2 -8564.866} C_VEL
LIN {X 0,Y 408.633,Z 732.854,A -85,B 0,C 180,E1 -8566.926,E2 -8566.926} C_VEL
LIN {X 0,Y 408.288,Z 738.413,A -85,B 0,C 180,E1 -8569.155,E2 -8569.155} C_VEL
LIN {X 0,Y 408.118,Z 742.175,A -85,B 0,C 180,E1 -8571.411,E2 -8571.411} C_VEL
LIN {X 0,Y 408.055,Z 744.119,A -85,B 0,C 180,E1 -8573.692,E2 -8573.692} C_VEL
LIN {X 0,Y 408.056,Z 744.351,A -85,B 0,C 180,E1 -8576.013,E2 -8576.013} C_VEL
LIN {X 0,Y 408.114,Z 742.658,A -85,B 0,C 180,E1 -8578.376,E2 -8578.376} C_VEL
LIN {X 0,Y 408.274,Z 739.319,A -85,B 0,C 180,E1 -8580.621,E2 -8580.621} C_VEL
LIN {X 0,Y 408.578,Z 734.395,A -85,B 0,C 180,E1 -8582.737,E2 -8582.737} C_VEL
LIN {X 0,Y 409.107,Z 727.572,A -85,B 0,C 180,E1 -8584.88,E2 -8584.88} C_VEL
LIN {X 0,Y 409.847,Z 719.188,A -85,B 0,C 180,E1 -8586.877,E2 -8586.877} C_VEL
LIN {X 0,Y 410.777,Z 709.377,A -85,B 0,C 180,E1 -8588.72,E2 -8588.72} C_VEL
LIN {X 0,Y 411.856,Z 698.132,A -85,B 0,C 180,E1 -8590.403,E2 -8590.403} C_VEL
LIN {X 0,Y 413.017,Z 685.395,A -85,B 0,C 180,E1 -8591.922,E2 -8591.922} C_VEL
LIN {X 0,Y 414.138,Z 672.032,A -85,B 0,C 180,E1 -8593.186,E2 -8593.186} C_VEL
LIN {X 0,Y 415.226,Z 656.9,A -85,B 0,C 180,E1 -8594.289,E2 -8594.289} C_VEL
LIN {X 0,Y 416.072,Z 641.531,A -85,B 0,C 180,E1 -8595.12,E2 -8595.12} C_VEL
LIN {X 0,Y 416.686,Z 624.56,A -85,B 0,C 180,E1 -8595.741,E2 -8595.741} C_VEL
LIN {X 0,Y 417.094,Z 601.073,A -85,B 0,C 180,E1 -8596.212,E2 -8596.212} C_VEL
LIN {X 0,Y 418.77,Z 491.392,A -85,B 0,C 180,E1 -8598.159,E2 -8598.159} C_VEL
LIN {X 0,Y 417.272,Z 478.572,A -85,B 0,C 180,E1 -8598.505,E2 -8598.505} C_VEL
LIN {X 0,Y 419.22,Z 435.152,A -85,B 0,C 180,E1 -8602.368,E2 -8602.368} C_VEL
LIN {X 0,Y 421.374,Z 390.604,A -85,B 0,C 180,E1 -8606.328,E2 -8606.328} C_VEL
LIN {X 0,Y 423.186,Z 346.815,A -85,B 0,C 180,E1 -8610.175,E2 -8610.175} C_VEL
LIN {X 0,Y 423.888,Z 325.31,A -85,B 0,C 180,E1 -8612.081,E2 -8612.081} C_VEL
LIN {X 0,Y 417.839,Z 306.895,A -85,B 0,C 180,E1 -8614.334,E2 -8614.334} C_VEL
LIN {X 0,Y 410.798,Z 289.054,A -85,B 0,C 180,E1 -8616.701,E2 -8616.701} C_VEL
LIN {X 0,Y 409.445,Z 285.747,A -85,B 0,C 180,E1 -8617.228,E2 -8617.228} C_VEL
LIN {X 0,Y 409.441,Z 285.48,A -85,B 0,C 180,E1 -8620.602,E2 -8620.602} C_VEL
LIN {X 0,Y 409.445,Z 285.474,A -85,B 0,C 180,E1 -8624.563,E2 -8624.563} C_VEL
LIN {X 0,Y 409.438,Z 285.488,A -85,B 0,C 180,E1 -8628.448,E2 -8628.448} C_VEL
LIN {X 0,Y 409.44,Z 285.487,A -85,B 0,C 180,E1 -8632.422,E2 -8632.422} C_VEL
LIN {X 0,Y 409.43,Z 285.483,A -85,B 0,C 180,E1 -8636.359,E2 -8636.359} C_VEL
LIN {X 0,Y 409.426,Z 285.486,A -85,B 0,C 180,E1 -8640.279,E2 -8640.279} C_VEL
LIN {X 0,Y 409.418,Z 285.482,A -85,B 0,C 180,E1 -8644.201,E2 -8644.201} C_VEL
LIN {X 0,Y 409.41,Z 285.486,A -85,B 0,C 180,E1 -8648.001,E2 -8648.001} C_VEL
LIN {X 0,Y 409.409,Z 285.486,A -85,B 0,C 180,E1 -8651.838,E2 -8651.838} C_VEL
LIN {X 0,Y 409.409,Z 285.48,A -85,B 0,C 180,E1 -8655.806,E2 -8655.806} C_VEL
LIN {X 0,Y 409.414,Z 285.483,A -85,B 0,C 180,E1 -8659.695,E2 -8659.695} C_VEL
LIN {X 0,Y 409.42,Z 285.484,A -85,B 0,C 180,E1 -8663.61,E2 -8663.61} C_VEL
LIN {X 0,Y 409.429,Z 285.481,A -85,B 0,C 180,E1 -8667.487,E2 -8667.487} C_VEL
LIN {X 0,Y 409.44,Z 285.481,A -85,B 0,C 180,E1 -8671.342,E2 -8671.342} C_VEL
LIN {X 0,Y 409.442,Z 285.484,A -85,B 0,C 180,E1 -8675.191,E2 -8675.191} C_VEL
LIN {X 0,Y 409.447,Z 285.483,A -85,B 0,C 180,E1 -8679.058,E2 -8679.058} C_VEL
LIN {X 0,Y 409.441,Z 285.482,A -85,B 0,C 180,E1 -8682.946,E2 -8682.946} C_VEL
LIN {X 0,Y 409.455,Z 285.752,A -85,B 0,C 180,E1 -8684.19,E2 -8684.19} C_VEL
LIN {X 0,Y 413.697,Z 295.947,A -85,B 0,C 180,E1 -8685.891,E2 -8685.891} C_VEL
LIN {X 0,Y 422.584,Z 317.111,A -85,B 0,C 180,E1 -8689.108,E2 -8689.108} C_VEL
LIN {X 0,Y 423.974,Z 319.962,A -85,B 0,C 180,E1 -8689.408,E2 -8689.408} C_VEL
LIN {X 0,Y 435.36,Z 340.774,A -85,B 0,C 180,E1 -8691,E2 -8691} C_VEL
LIN {X 0,Y 436.163,Z 348.636,A -85,B 0,C 180,E1 -8691.257,E2 -8691.257} C_VEL
LIN {X 0,Y 429.865,Z 532.714,A -85,B 0,C 180,E1 -8694.867,E2 -8694.867} C_VEL
LIN {X 0,Y 428.331,Z 578.448,A -85,B 0,C 180,E1 -8695.789,E2 -8695.789} C_VEL
LIN {X 0,Y 427.043,Z 599.463,A -85,B 0,C 180,E1 -8696.444,E2 -8696.444} C_VEL
LIN {X 0,Y 425.338,Z 620.362,A -85,B 0,C 180,E1 -8697.353,E2 -8697.353} C_VEL
LIN {X 0,Y 423.343,Z 641.074,A -85,B 0,C 180,E1 -8698.538,E2 -8698.538} C_VEL
LIN {X 0,Y 421.182,Z 660.578,A -85,B 0,C 180,E1 -8699.943,E2 -8699.943} C_VEL
LIN {X 0,Y 418.95,Z 678.998,A -85,B 0,C 180,E1 -8701.57,E2 -8701.57} C_VEL
LIN {X 0,Y 416.812,Z 695.719,A -85,B 0,C 180,E1 -8703.349,E2 -8703.349} C_VEL
LIN {X 0,Y 414.743,Z 711.551,A -85,B 0,C 180,E1 -8705.352,E2 -8705.352} C_VEL
LIN {X 0,Y 412.908,Z 725.909,A -85,B 0,C 180,E1 -8707.507,E2 -8707.507} C_VEL
LIN {X 0,Y 411.253,Z 739.579,A -85,B 0,C 180,E1 -8709.954,E2 -8709.954} C_VEL
LIN {X 0,Y 409.975,Z 751.287,A -85,B 0,C 180,E1 -8712.473,E2 -8712.473} C_VEL
LIN {X 0,Y 409.08,Z 760.974,A -85,B 0,C 180,E1 -8714.986,E2 -8714.986} C_VEL
LIN {X 0,Y 408.457,Z 769.464,A -85,B 0,C 180,E1 -8717.705,E2 -8717.705} C_VEL
LIN {X 0,Y 408.127,Z 776.005,A -85,B 0,C 180,E1 -8720.412,E2 -8720.412} C_VEL
LIN {X 0,Y 408.001,Z 780.825,A -85,B 0,C 180,E1 -8723.105,E2 -8723.105} C_VEL
LIN {X 0,Y 407.975,Z 784.153,A -85,B 0,C 180,E1 -8725.926,E2 -8725.926} C_VEL
LIN {X 0,Y 407.977,Z 785.727,A -85,B 0,C 180,E1 -8728.597,E2 -8728.597} C_VEL
LIN {X 0,Y 407.987,Z 785.708,A -85,B 0,C 180,E1 -8731.125,E2 -8731.125} C_VEL
LIN {X 0,Y 407.981,Z 784.184,A -85,B 0,C 180,E1 -8733.796,E2 -8733.796} C_VEL
LIN {X 0,Y 408,Z 781.107,A -85,B 0,C 180,E1 -8736.474,E2 -8736.474} C_VEL
LIN {X 0,Y 408.103,Z 776.347,A -85,B 0,C 180,E1 -8739.165,E2 -8739.165} C_VEL
LIN {X 0,Y 408.363,Z 770.157,A -85,B 0,C 180,E1 -8741.727,E2 -8741.727} C_VEL
LIN {X 0,Y 408.894,Z 761.726,A -85,B 0,C 180,E1 -8744.46,E2 -8744.46} C_VEL
LIN {X 0,Y 409.7,Z 751.884,A -85,B 0,C 180,E1 -8747.03,E2 -8747.03} C_VEL
LIN {X 0,Y 410.808,Z 740.532,A -85,B 0,C 180,E1 -8749.479,E2 -8749.479} C_VEL
LIN {X 0,Y 412.193,Z 727.752,A -85,B 0,C 180,E1 -8751.787,E2 -8751.787} C_VEL
LIN {X 0,Y 413.956,Z 712.453,A -85,B 0,C 180,E1 -8754.093,E2 -8754.093} C_VEL
LIN {X 0,Y 415.898,Z 695.878,A -85,B 0,C 180,E1 -8756.179,E2 -8756.179} C_VEL
LIN {X 0,Y 417.908,Z 678.404,A -85,B 0,C 180,E1 -8758.013,E2 -8758.013} C_VEL
LIN {X 0,Y 419.918,Z 660.099,A -85,B 0,C 180,E1 -8759.61,E2 -8759.61} C_VEL
LIN {X 0,Y 421.825,Z 641.387,A -85,B 0,C 180,E1 -8760.956,E2 -8760.956} C_VEL
LIN {X 0,Y 423.642,Z 621.478,A -85,B 0,C 180,E1 -8762.116,E2 -8762.116} C_VEL
LIN {X 0,Y 425.313,Z 600.478,A -85,B 0,C 180,E1 -8763.069,E2 -8763.069} C_VEL
LIN {X 0,Y 426.713,Z 578.887,A -85,B 0,C 180,E1 -8763.785,E2 -8763.785} C_VEL
LIN {X 0,Y 428.431,Z 536.993,A -85,B 0,C 180,E1 -8764.718,E2 -8764.718} C_VEL
LIN {X 0,Y 431.798,Z 465.751,A -85,B 0,C 180,E1 -8766.345,E2 -8766.345} C_VEL
LIN {X 0,Y 436.632,Z 395.58,A -85,B 0,C 180,E1 -8768.124,E2 -8768.124} C_VEL
LIN {X 0,Y 440.822,Z 347.159,A -85,B 0,C 180,E1 -8769.462,E2 -8769.462} C_VEL
LIN {X 0,Y 440.653,Z 343.03,A -85,B 0,C 180,E1 -8769.693,E2 -8769.693} C_VEL
LIN {X 0,Y 437.475,Z 336.184,A -85,B 0,C 180,E1 -8770.693,E2 -8770.693} C_VEL
LIN {X 0,Y 434.845,Z 331.426,A -85,B 0,C 180,E1 -8771.646,E2 -8771.646} C_VEL
LIN {X 0,Y 432.59,Z 327.549,A -85,B 0,C 180,E1 -8772.693,E2 -8772.693} C_VEL
LIN {X 0,Y 431.952,Z 325.727,A -85,B 0,C 180,E1 -8773.615,E2 -8773.615} C_VEL
LIN {X 0,Y 431.536,Z 323.543,A -85,B 0,C 180,E1 -8775.409,E2 -8775.409} C_VEL
LIN {X 0,Y 431.432,Z 323.706,A -85,B 0,C 180,E1 -8776.89,E2 -8776.89} C_VEL
LIN {X 0,Y 431.955,Z 326.581,A -85,B 0,C 180,E1 -8779.076,E2 -8779.076} C_VEL
LIN {X 0,Y 433.064,Z 331.226,A -85,B 0,C 180,E1 -8780.928,E2 -8780.928} C_VEL
LIN {X 0,Y 434.094,Z 335.275,A -85,B 0,C 180,E1 -8782.05,E2 -8782.05} C_VEL
LIN {X 0,Y 437.443,Z 343.141,A -85,B 0,C 180,E1 -8783.432,E2 -8783.432} C_VEL
LIN {X 0,Y 438.732,Z 362.342,A -85,B 0,C 180,E1 -8784.73,E2 -8784.73} C_VEL
LIN {X 0,Y 439.181,Z 375.076,A -85,B 0,C 180,E1 -8785.413,E2 -8785.413} C_VEL
LIN {X 0,Y 432.067,Z 453.004,A -85,B 0,C 180,E1 -8787.563,E2 -8787.563} C_VEL
LIN {X 0,Y 427.349,Z 524.988,A -85,B 0,C 180,E1 -8789.424,E2 -8789.424} C_VEL
LIN {X 0,Y 425.041,Z 568.087,A -85,B 0,C 180,E1 -8790.514,E2 -8790.514} C_VEL
LIN {X 0,Y 423.582,Z 588.718,A -85,B 0,C 180,E1 -8791.292,E2 -8791.292} C_VEL
LIN {X 0,Y 421.977,Z 607.641,A -85,B 0,C 180,E1 -8792.251,E2 -8792.251} C_VEL
LIN {X 0,Y 420.222,Z 625.834,A -85,B 0,C 180,E1 -8793.429,E2 -8793.429} C_VEL
LIN {X 0,Y 418.356,Z 643.232,A -85,B 0,C 180,E1 -8794.824,E2 -8794.824} C_VEL
LIN {X 0,Y 416.456,Z 659.71,A -85,B 0,C 180,E1 -8796.438,E2 -8796.438} C_VEL
LIN {X 0,Y 414.595,Z 675.147,A -85,B 0,C 180,E1 -8798.273,E2 -8798.273} C_VEL
LIN {X 0,Y 412.85,Z 689.394,A -85,B 0,C 180,E1 -8800.328,E2 -8800.328} C_VEL
LIN {X 0,Y 411.39,Z 701.591,A -85,B 0,C 180,E1 -8802.46,E2 -8802.46} C_VEL
LIN {X 0,Y 410.189,Z 712.307,A -85,B 0,C 180,E1 -8804.737,E2 -8804.737} C_VEL
LIN {X 0,Y 409.272,Z 721.526,A -85,B 0,C 180,E1 -8807.155,E2 -8807.155} C_VEL
LIN {X 0,Y 408.634,Z 729.185,A -85,B 0,C 180,E1 -8809.711,E2 -8809.711} C_VEL
LIN {X 0,Y 408.26,Z 734.944,A -85,B 0,C 180,E1 -8812.259,E2 -8812.259} C_VEL
LIN {X 0,Y 408.085,Z 738.969,A -85,B 0,C 180,E1 -8814.799,E2 -8814.799} C_VEL
LIN {X 0,Y 408.009,Z 741.429,A -85,B 0,C 180,E1 -8817.472,E2 -8817.472} C_VEL
LIN {X 0,Y 407.997,Z 742.14,A -85,B 0,C 180,E1 -8820.141,E2 -8820.141} C_VEL
LIN {X 0,Y 408.003,Z 741.115,A -85,B 0,C 180,E1 -8822.81,E2 -8822.81} C_VEL
LIN {X 0,Y 408.067,Z 738.34,A -85,B 0,C 180,E1 -8825.484,E2 -8825.484} C_VEL
LIN {X 0,Y 408.239,Z 734.039,A -85,B 0,C 180,E1 -8828.025,E2 -8828.025} C_VEL
LIN {X 0,Y 408.607,Z 727.988,A -85,B 0,C 180,E1 -8830.576,E2 -8830.576} C_VEL
LIN {X 0,Y 409.246,Z 720.031,A -85,B 0,C 180,E1 -8833.134,E2 -8833.134} C_VEL
LIN {X 0,Y 410.177,Z 710.522,A -85,B 0,C 180,E1 -8835.554,E2 -8835.554} C_VEL
LIN {X 0,Y 411.391,Z 699.517,A -85,B 0,C 180,E1 -8837.833,E2 -8837.833} C_VEL
LIN {X 0,Y 412.919,Z 686.635,A -85,B 0,C 180,E1 -8840.027,E2 -8840.027} C_VEL
LIN {X 0,Y 414.575,Z 673.027,A -85,B 0,C 180,E1 -8841.952,E2 -8841.952} C_VEL
LIN {X 0,Y 416.382,Z 658.041,A -85,B 0,C 180,E1 -8843.718,E2 -8843.718} C_VEL
LIN {X 0,Y 418.203,Z 642.211,A -85,B 0,C 180,E1 -8845.263,E2 -8845.263} C_VEL
LIN {X 0,Y 420.071,Z 624.636,A -85,B 0,C 180,E1 -8846.662,E2 -8846.662} C_VEL
LIN {X 0,Y 421.795,Z 606.079,A -85,B 0,C 180,E1 -8847.839,E2 -8847.839} C_VEL
LIN {X 0,Y 423.294,Z 587.005,A -85,B 0,C 180,E1 -8848.769,E2 -8848.769} C_VEL
LIN {X 0,Y 424.503,Z 567.385,A -85,B 0,C 180,E1 -8849.462,E2 -8849.462} C_VEL
LIN {X 0,Y 425.458,Z 542.817,A -85,B 0,C 180,E1 -8850.019,E2 -8850.019} C_VEL
LIN {X 0,Y 431.126,Z 371.276,A -85,B 0,C 180,E1 -8853.46,E2 -8853.46} C_VEL
LIN {X 0,Y 426.483,Z 339.985,A -85,B 0,C 180,E1 -8854.653,E2 -8854.653} C_VEL
LIN {X 0,Y 427.084,Z 332.903,A -85,B 0,C 180,E1 -8855.374,E2 -8855.374} C_VEL
LIN {X 0,Y 420.829,Z 314.961,A -85,B 0,C 180,E1 -8858.035,E2 -8858.035} C_VEL
LIN {X 0,Y 413.241,Z 295.326,A -85,B 0,C 180,E1 -8861.193,E2 -8861.193} C_VEL
LIN {X 0,Y 409.469,Z 285.685,A -85,B 0,C 180,E1 -8862.889,E2 -8862.889} C_VEL
LIN {X 0,Y 409.437,Z 285.476,A -85,B 0,C 180,E1 -8866.697,E2 -8866.697} C_VEL
LIN {X 0,Y 409.444,Z 285.483,A -85,B 0,C 180,E1 -8870.585,E2 -8870.585} C_VEL
LIN {X 0,Y 409.438,Z 285.487,A -85,B 0,C 180,E1 -8874.464,E2 -8874.464} C_VEL
LIN {X 0,Y 409.443,Z 285.486,A -85,B 0,C 180,E1 -8878.328,E2 -8878.328} C_VEL
LIN {X 0,Y 409.443,Z 285.478,A -85,B 0,C 180,E1 -8882.196,E2 -8882.196} C_VEL
LIN {X 0,Y 409.444,Z 285.474,A -85,B 0,C 180,E1 -8886.084,E2 -8886.084} C_VEL
LIN {X 0,Y 409.404,Z 285.475,A -85,B 0,C 180,E1 -8889.117,E2 -8889.117} C_VEL
LIN {X 0,Y 408.633,Z 286.013,A -85,B 0,C 180,E1 -8890.167,E2 -8890.167} C_VEL
LIN {X 0,Y 406.513,Z 288.248,A -85,B 0,C 180,E1 -8891.471,E2 -8891.471} C_VEL
LIN {X 0,Y 405.109,Z 291.765,A -85,B 0,C 180,E1 -8892.542,E2 -8892.542} C_VEL
LIN {X 0,Y 405.189,Z 295.467,A -85,B 0,C 180,E1 -8893.257,E2 -8893.257} C_VEL
LIN {X 0,Y 405.561,Z 296.905,A -85,B 0,C 180,E1 -8893.465,E2 -8893.465} C_VEL
LIN {X 0,Y 412.964,Z 317.049,A -85,B 0,C 180,E1 -8896.145,E2 -8896.145} C_VEL
LIN {X 0,Y 417.029,Z 329.886,A -85,B 0,C 180,E1 -8897.748,E2 -8897.748} C_VEL
LIN {X 0,Y 414.96,Z 371.575,A -85,B 0,C 180,E1 -8901.547,E2 -8901.547} C_VEL
LIN {X 0,Y 412.836,Z 411.688,A -85,B 0,C 180,E1 -8905.206,E2 -8905.206} C_VEL
LIN {X 0,Y 410.672,Z 454.282,A -85,B 0,C 180,E1 -8909.072,E2 -8909.072} C_VEL
LIN {X 0,Y 409.505,Z 478.654,A -85,B 0,C 180,E1 -8911.266,E2 -8911.266} C_VEL
LIN {X 0,Y 411.224,Z 495.271,A -85,B 0,C 180,E1 -8911.685,E2 -8911.685} C_VEL
LIN {X 0,Y 409.029,Z 621.938,A -85,B 0,C 180,E1 -8913.976,E2 -8913.976} C_VEL
LIN {X 0,Y 408.474,Z 637.95,A -85,B 0,C 180,E1 -8914.522,E2 -8914.522} C_VEL
LIN {X 0,Y 407.614,Z 654.079,A -85,B 0,C 180,E1 -8915.347,E2 -8915.347} C_VEL
LIN {X 0,Y 406.598,Z 668.45,A -85,B 0,C 180,E1 -8916.352,E2 -8916.352} C_VEL
LIN {X 0,Y 405.397,Z 682.78,A -85,B 0,C 180,E1 -8917.652,E2 -8917.652} C_VEL
LIN {X 0,Y 404.228,Z 695.407,A -85,B 0,C 180,E1 -8919.107,E2 -8919.107} C_VEL
LIN {X 0,Y 403.037,Z 707.547,A -85,B 0,C 180,E1 -8920.866,E2 -8920.866} C_VEL
LIN {X 0,Y 402.083,Z 717.305,A -85,B 0,C 180,E1 -8922.639,E2 -8922.639} C_VEL
LIN {X 0,Y 401.228,Z 726.581,A -85,B 0,C 180,E1 -8924.781,E2 -8924.781} C_VEL
LIN {X 0,Y 400.68,Z 733.373,A -85,B 0,C 180,E1 -8926.824,E2 -8926.824} C_VEL
LIN {X 0,Y 400.312,Z 738.903,A -85,B 0,C 180,E1 -8929.097,E2 -8929.097} C_VEL
LIN {X 0,Y 400.132,Z 742.614,A -85,B 0,C 180,E1 -8931.395,E2 -8931.395} C_VEL
LIN {X 0,Y 400.064,Z 744.585,A -85,B 0,C 180,E1 -8933.832,E2 -8933.832} C_VEL
LIN {X 0,Y 400.066,Z 744.723,A -85,B 0,C 180,E1 -8936.093,E2 -8936.093} C_VEL
LIN {X 0,Y 400.134,Z 742.993,A -85,B 0,C 180,E1 -8938.505,E2 -8938.505} C_VEL
LIN {X 0,Y 400.315,Z 739.607,A -85,B 0,C 180,E1 -8940.796,E2 -8940.796} C_VEL
LIN {X 0,Y 400.683,Z 734.177,A -85,B 0,C 180,E1 -8943.124,E2 -8943.124} C_VEL
LIN {X 0,Y 401.239,Z 727.638,A -85,B 0,C 180,E1 -8945.178,E2 -8945.178} C_VEL
LIN {X 0,Y 402.072,Z 718.864,A -85,B 0,C 180,E1 -8947.271,E2 -8947.271} C_VEL
LIN {X 0,Y 403.085,Z 708.931,A -85,B 0,C 180,E1 -8949.143,E2 -8949.143} C_VEL
LIN {X 0,Y 404.242,Z 697.485,A -85,B 0,C 180,E1 -8950.848,E2 -8950.848} C_VEL
LIN {X 0,Y 405.505,Z 684.436,A -85,B 0,C 180,E1 -8952.404,E2 -8952.404} C_VEL
LIN {X 0,Y 406.721,Z 670.306,A -85,B 0,C 180,E1 -8953.717,E2 -8953.717} C_VEL
LIN {X 0,Y 407.821,Z 655.569,A -85,B 0,C 180,E1 -8954.777,E2 -8954.777} C_VEL
LIN {X 0,Y 408.703,Z 639.406,A -85,B 0,C 180,E1 -8955.621,E2 -8955.621} C_VEL
LIN {X 0,Y 409.283,Z 623.246,A -85,B 0,C 180,E1 -8956.19,E2 -8956.19} C_VEL
LIN {X 0,Y 410.285,Z 565.115,A -85,B 0,C 180,E1 -8957.271,E2 -8957.271} C_VEL
LIN {X 0,Y 411.454,Z 492.273,A -85,B 0,C 180,E1 -8958.596,E2 -8958.596} C_VEL
LIN {X 0,Y 409.896,Z 478.596,A -85,B 0,C 180,E1 -8958.991,E2 -8958.991} C_VEL
LIN {X 0,Y 411.938,Z 436.084,A -85,B 0,C 180,E1 -8962.815,E2 -8962.815} C_VEL
LIN {X 0,Y 413.964,Z 395.766,A -85,B 0,C 180,E1 -8966.419,E2 -8966.419} C_VEL
LIN {X 0,Y 415.691,Z 358.54,A -85,B 0,C 180,E1 -8969.74,E2 -8969.74} C_VEL
LIN {X 0,Y 416.909,Z 328.405,A -85,B 0,C 180,E1 -8972.427,E2 -8972.427} C_VEL
LIN {X 0,Y 411.048,Z 310.536,A -85,B 0,C 180,E1 -8974.651,E2 -8974.651} C_VEL
LIN {X 0,Y 404.238,Z 293.317,A -85,B 0,C 180,E1 -8976.995,E2 -8976.995} C_VEL
LIN {X 0,Y 401.548,Z 286.939,A -85,B 0,C 180,E1 -8977.952,E2 -8977.952} C_VEL
LIN {X 0,Y 401.507,Z 286.466,A -85,B 0,C 180,E1 -8978.373,E2 -8978.373} C_VEL
LIN {X 0,Y 401.494,Z 286.468,A -85,B 0,C 180,E1 -8982.312,E2 -8982.312} C_VEL
LIN {X 0,Y 401.49,Z 286.478,A -85,B 0,C 180,E1 -8986.217,E2 -8986.217} C_VEL
LIN {X 0,Y 401.479,Z 286.477,A -85,B 0,C 180,E1 -8990.105,E2 -8990.105} C_VEL
LIN {X 0,Y 401.475,Z 286.473,A -85,B 0,C 180,E1 -8993.995,E2 -8993.995} C_VEL
LIN {X 0,Y 401.468,Z 286.477,A -85,B 0,C 180,E1 -8997.859,E2 -8997.859} C_VEL
LIN {X 0,Y 401.468,Z 286.472,A -85,B 0,C 180,E1 -9001.712,E2 -9001.712} C_VEL
LIN {X 0,Y 401.469,Z 286.475,A -85,B 0,C 180,E1 -9005.717,E2 -9005.717} C_VEL
LIN {X 0,Y 401.473,Z 286.469,A -85,B 0,C 180,E1 -9009.605,E2 -9009.605} C_VEL
LIN {X 0,Y 401.477,Z 286.472,A -85,B 0,C 180,E1 -9013.538,E2 -9013.538} C_VEL
LIN {X 0,Y 401.488,Z 286.473,A -85,B 0,C 180,E1 -9017.388,E2 -9017.388} C_VEL
LIN {X 0,Y 401.493,Z 286.468,A -85,B 0,C 180,E1 -9021.354,E2 -9021.354} C_VEL
LIN {X 0,Y 401.496,Z 286.472,A -85,B 0,C 180,E1 -9025.318,E2 -9025.318} C_VEL
LIN {X 0,Y 401.509,Z 286.468,A -85,B 0,C 180,E1 -9029.215,E2 -9029.215} C_VEL
LIN {X 0,Y 401.502,Z 286.472,A -85,B 0,C 180,E1 -9033.22,E2 -9033.22} C_VEL
LIN {X 0,Y 401.504,Z 286.472,A -85,B 0,C 180,E1 -9037.238,E2 -9037.238} C_VEL
LIN {X 0,Y 401.508,Z 286.47,A -85,B 0,C 180,E1 -9041.234,E2 -9041.234} C_VEL
LIN {X 0,Y 401.541,Z 286.736,A -85,B 0,C 180,E1 -9043.336,E2 -9043.336} C_VEL
LIN {X 0,Y 404.51,Z 293.868,A -85,B 0,C 180,E1 -9044.586,E2 -9044.586} C_VEL
LIN {X 0,Y 413.46,Z 315.115,A -85,B 0,C 180,E1 -9047.946,E2 -9047.946} C_VEL
LIN {X 0,Y 415.177,Z 319.194,A -85,B 0,C 180,E1 -9048.501,E2 -9048.501} C_VEL
LIN {X 0,Y 428.834,Z 343.693,A -85,B 0,C 180,E1 -9050.458,E2 -9050.458} C_VEL
LIN {X 0,Y 429.555,Z 349.719,A -85,B 0,C 180,E1 -9050.671,E2 -9050.671} C_VEL
LIN {X 0,Y 422.825,Z 534.371,A -85,B 0,C 180,E1 -9054.374,E2 -9054.374} C_VEL
LIN {X 0,Y 421.256,Z 578.403,A -85,B 0,C 180,E1 -9055.282,E2 -9055.282} C_VEL
LIN {X 0,Y 419.91,Z 599.404,A -85,B 0,C 180,E1 -9055.95,E2 -9055.95} C_VEL
LIN {X 0,Y 418.113,Z 620.428,A -85,B 0,C 180,E1 -9056.88,E2 -9056.88} C_VEL
LIN {X 0,Y 416.039,Z 641.087,A -85,B 0,C 180,E1 -9058.083,E2 -9058.083} C_VEL
LIN {X 0,Y 413.78,Z 660.538,A -85,B 0,C 180,E1 -9059.508,E2 -9059.508} C_VEL
LIN {X 0,Y 411.454,Z 678.932,A -85,B 0,C 180,E1 -9061.162,E2 -9061.162} C_VEL
LIN {X 0,Y 409.219,Z 695.653,A -85,B 0,C 180,E1 -9062.972,E2 -9062.972} C_VEL
LIN {X 0,Y 407.127,Z 710.957,A -85,B 0,C 180,E1 -9064.937,E2 -9064.937} C_VEL
LIN {X 0,Y 405.255,Z 724.947,A -85,B 0,C 180,E1 -9067.059,E2 -9067.059} C_VEL
LIN {X 0,Y 403.582,Z 738.014,A -85,B 0,C 180,E1 -9069.405,E2 -9069.405} C_VEL
LIN {X 0,Y 402.229,Z 749.671,A -85,B 0,C 180,E1 -9071.899,E2 -9071.899} C_VEL
LIN {X 0,Y 401.216,Z 759.861,A -85,B 0,C 180,E1 -9074.537,E2 -9074.537} C_VEL
LIN {X 0,Y 400.52,Z 768.473,A -85,B 0,C 180,E1 -9077.311,E2 -9077.311} C_VEL
LIN {X 0,Y 400.173,Z 774.86,A -85,B 0,C 180,E1 -9079.929,E2 -9079.929} C_VEL
LIN {X 0,Y 400.004,Z 779.926,A -85,B 0,C 180,E1 -9082.678,E2 -9082.678} C_VEL
LIN {X 0,Y 399.977,Z 783.361,A -85,B 0,C 180,E1 -9085.413,E2 -9085.413} C_VEL
LIN {X 0,Y 399.99,Z 785.136,A -85,B 0,C 180,E1 -9088.139,E2 -9088.139} C_VEL
LIN {X 0,Y 400.001,Z 785.331,A -85,B 0,C 180,E1 -9090.861,E2 -9090.861} C_VEL
LIN {X 0,Y 399.986,Z 783.985,A -85,B 0,C 180,E1 -9093.584,E2 -9093.584} C_VEL
LIN {X 0,Y 400.003,Z 781.06,A -85,B 0,C 180,E1 -9096.316,E2 -9096.316} C_VEL
LIN {X 0,Y 400.1,Z 776.391,A -85,B 0,C 180,E1 -9099.06,E2 -9099.06} C_VEL
LIN {X 0,Y 400.375,Z 769.983,A -85,B 0,C 180,E1 -9101.818,E2 -9101.818} C_VEL
LIN {X 0,Y 400.935,Z 761.544,A -85,B 0,C 180,E1 -9104.626,E2 -9104.626} C_VEL
LIN {X 0,Y 401.776,Z 751.827,A -85,B 0,C 180,E1 -9107.227,E2 -9107.227} C_VEL
LIN {X 0,Y 402.944,Z 740.542,A -85,B 0,C 180,E1 -9109.724,E2 -9109.724} C_VEL
LIN {X 0,Y 404.402,Z 727.805,A -85,B 0,C 180,E1 -9112.076,E2 -9112.076} C_VEL
LIN {X 0,Y 406.132,Z 713.597,A -85,B 0,C 180,E1 -9114.278,E2 -9114.278} C_VEL
LIN {X 0,Y 408.074,Z 697.927,A -85,B 0,C 180,E1 -9116.328,E2 -9116.328} C_VEL
LIN {X 0,Y 410.113,Z 681.403,A -85,B 0,C 180,E1 -9118.15,E2 -9118.15} C_VEL
LIN {X 0,Y 412.357,Z 662.488,A -85,B 0,C 180,E1 -9119.888,E2 -9119.888} C_VEL
LIN {X 0,Y 414.568,Z 642.382,A -85,B 0,C 180,E1 -9121.397,E2 -9121.397} C_VEL
LIN {X 0,Y 416.592,Z 621.862,A -85,B 0,C 180,E1 -9122.633,E2 -9122.633} C_VEL
LIN {X 0,Y 418.438,Z 600.512,A -85,B 0,C 180,E1 -9123.63,E2 -9123.63} C_VEL
LIN {X 0,Y 419.993,Z 578.499,A -85,B 0,C 180,E1 -9124.384,E2 -9124.384} C_VEL
LIN {X 0,Y 424.822,Z 481.64,A -85,B 0,C 180,E1 -9126.663,E2 -9126.663} C_VEL
LIN {X 0,Y 429.874,Z 412.916,A -85,B 0,C 180,E1 -9128.456,E2 -9128.456} C_VEL
LIN {X 0,Y 436.14,Z 349.307,A -85,B 0,C 180,E1 -9130.262,E2 -9130.262} C_VEL
LIN {X 0,Y 435.987,Z 347.106,A -85,B 0,C 180,E1 -9130.414,E2 -9130.414} C_VEL
LIN {X 0,Y 433.137,Z 340.697,A -85,B 0,C 180,E1 -9131.478,E2 -9131.478} C_VEL
LIN {X 0,Y 430.138,Z 335.241,A -85,B 0,C 180,E1 -9132.83,E2 -9132.83} C_VEL
LIN {X 0,Y 428.517,Z 332.86,A -85,B 0,C 180,E1 -9133.768,E2 -9133.768} C_VEL
LIN {X 0,Y 426.957,Z 330.107,A -85,B 0,C 180,E1 -9135.369,E2 -9135.369} C_VEL
LIN {X 0,Y 426.709,Z 330.165,A -85,B 0,C 180,E1 -9136.827,E2 -9136.827} C_VEL
LIN {X 0,Y 427.112,Z 332.871,A -85,B 0,C 180,E1 -9138.921,E2 -9138.921} C_VEL
LIN {X 0,Y 428.732,Z 337.025,A -85,B 0,C 180,E1 -9140.377,E2 -9140.377} C_VEL
LIN {X 0,Y 431.191,Z 342.596,A -85,B 0,C 180,E1 -9141.774,E2 -9141.774} C_VEL
LIN {X 0,Y 433.391,Z 348.399,A -85,B 0,C 180,E1 -9142.793,E2 -9142.793} C_VEL
LIN {X 0,Y 434.095,Z 366.894,A -85,B 0,C 180,E1 -9144.072,E2 -9144.072} C_VEL
LIN {X 0,Y 434.18,Z 376.926,A -85,B 0,C 180,E1 -9144.618,E2 -9144.618} C_VEL
LIN {X 0,Y 426.359,Z 453.054,A -85,B 0,C 180,E1 -9146.811,E2 -9146.811} C_VEL
LIN {X 0,Y 421.045,Z 524.214,A -85,B 0,C 180,E1 -9148.743,E2 -9148.743} C_VEL
LIN {X 0,Y 418.334,Z 568.989,A -85,B 0,C 180,E1 -9149.933,E2 -9149.933} C_VEL
LIN {X 0,Y 416.746,Z 589.436,A -85,B 0,C 180,E1 -9150.733,E2 -9150.733} C_VEL
LIN {X 0,Y 414.927,Z 609.187,A -85,B 0,C 180,E1 -9151.771,E2 -9151.771} C_VEL
LIN {X 0,Y 412.905,Z 628.546,A -85,B 0,C 180,E1 -9153.075,E2 -9153.075} C_VEL
LIN {X 0,Y 410.899,Z 645.811,A -85,B 0,C 180,E1 -9154.527,E2 -9154.527} C_VEL
LIN {X 0,Y 408.864,Z 662.153,A -85,B 0,C 180,E1 -9156.203,E2 -9156.203} C_VEL
LIN {X 0,Y 406.908,Z 677.187,A -85,B 0,C 180,E1 -9158.069,E2 -9158.069} C_VEL
LIN {X 0,Y 405.129,Z 690.8,A -85,B 0,C 180,E1 -9160.106,E2 -9160.106} C_VEL
LIN {X 0,Y 403.603,Z 702.744,A -85,B 0,C 180,E1 -9162.26,E2 -9162.26} C_VEL
LIN {X 0,Y 402.335,Z 713.337,A -85,B 0,C 180,E1 -9164.579,E2 -9164.579} C_VEL
LIN {X 0,Y 401.364,Z 722.444,A -85,B 0,C 180,E1 -9167.044,E2 -9167.044} C_VEL
LIN {X 0,Y 400.714,Z 729.647,A -85,B 0,C 180,E1 -9169.506,E2 -9169.506} C_VEL
LIN {X 0,Y 400.306,Z 735.408,A -85,B 0,C 180,E1 -9172.104,E2 -9172.104} C_VEL
LIN {X 0,Y 400.109,Z 739.43,A -85,B 0,C 180,E1 -9174.695,E2 -9174.695} C_VEL
LIN {X 0,Y 400.024,Z 741.88,A -85,B 0,C 180,E1 -9177.422,E2 -9177.422} C_VEL
LIN {X 0,Y 400.01,Z 742.584,A -85,B 0,C 180,E1 -9180.001,E2 -9180.001} C_VEL
LIN {X 0,Y 400.014,Z 741.619,A -85,B 0,C 180,E1 -9182.723,E2 -9182.723} C_VEL
LIN {X 0,Y 400.081,Z 738.898,A -85,B 0,C 180,E1 -9185.45,E2 -9185.45} C_VEL
LIN {X 0,Y 400.275,Z 734.348,A -85,B 0,C 180,E1 -9188.186,E2 -9188.186} C_VEL
LIN {X 0,Y 400.673,Z 728.235,A -85,B 0,C 180,E1 -9190.788,E2 -9190.788} C_VEL
LIN {X 0,Y 401.363,Z 720.196,A -85,B 0,C 180,E1 -9193.396,E2 -9193.396} C_VEL
LIN {X 0,Y 402.36,Z 710.601,A -85,B 0,C 180,E1 -9195.864,E2 -9195.864} C_VEL
LIN {X 0,Y 403.655,Z 699.494,A -85,B 0,C 180,E1 -9198.187,E2 -9198.187} C_VEL
LIN {X 0,Y 405.226,Z 686.896,A -85,B 0,C 180,E1 -9200.36,E2 -9200.36} C_VEL
LIN {X 0,Y 407.024,Z 672.753,A -85,B 0,C 180,E1 -9202.381,E2 -9202.381} C_VEL
LIN {X 0,Y 408.929,Z 657.613,A -85,B 0,C 180,E1 -9204.177,E2 -9204.177} C_VEL
LIN {X 0,Y 410.907,Z 641.043,A -85,B 0,C 180,E1 -9205.798,E2 -9205.798} C_VEL
LIN {X 0,Y 412.803,Z 623.895,A -85,B 0,C 180,E1 -9207.167,E2 -9207.167} C_VEL
LIN {X 0,Y 414.534,Z 606.056,A -85,B 0,C 180,E1 -9208.31,E2 -9208.31} C_VEL
LIN {X 0,Y 416.106,Z 586.84,A -85,B 0,C 180,E1 -9209.259,E2 -9209.259} C_VEL
LIN {X 0,Y 417.393,Z 566.886,A -85,B 0,C 180,E1 -9209.97,E2 -9209.97} C_VEL
LIN {X 0,Y 418.498,Z 538.975,A -85,B 0,C 180,E1 -9210.603,E2 -9210.603} C_VEL
LIN {X 0,Y 424.371,Z 372.403,A -85,B 0,C 180,E1 -9214.027,E2 -9214.027} C_VEL
LIN {X 0,Y 419.632,Z 339.846,A -85,B 0,C 180,E1 -9215.297,E2 -9215.297} C_VEL
LIN {X 0,Y 419.936,Z 335.776,A -85,B 0,C 180,E1 -9215.715,E2 -9215.715} C_VEL
LIN {X 0,Y 413.636,Z 317.721,A -85,B 0,C 180,E1 -9218.445,E2 -9218.445} C_VEL
LIN {X 0,Y 406.443,Z 299.158,A -85,B 0,C 180,E1 -9221.488,E2 -9221.488} C_VEL
LIN {X 0,Y 401.52,Z 286.668,A -85,B 0,C 180,E1 -9223.705,E2 -9223.705} C_VEL
LIN {X 0,Y 401.5,Z 286.469,A -85,B 0,C 180,E1 -9227.554,E2 -9227.554} C_VEL
LIN {X 0,Y 401.505,Z 286.472,A -85,B 0,C 180,E1 -9231.495,E2 -9231.495} C_VEL
LIN {X 0,Y 401.499,Z 286.47,A -85,B 0,C 180,E1 -9235.518,E2 -9235.518} C_VEL
LIN {X 0,Y 401.497,Z 286.462,A -85,B 0,C 180,E1 -9239.504,E2 -9239.504} C_VEL
LIN {X 0,Y 401.484,Z 286.474,A -85,B 0,C 180,E1 -9243.389,E2 -9243.389} C_VEL
LIN {X 0,Y 401.476,Z 286.476,A -85,B 0,C 180,E1 -9247.292,E2 -9247.292} C_VEL
LIN {X 0,Y 401.462,Z 286.47,A -85,B 0,C 180,E1 -9251.159,E2 -9251.159} C_VEL
LIN {X 0,Y 401.541,Z 286.773,A -85,B 0,C 180,E1 -9251.995,E2 -9251.995} C_VEL
LIN {X 0,Y 404.764,Z 295.056,A -85,B 0,C 180,E1 -9253.2,E2 -9253.2} C_VEL
LIN {X 0,Y 405.561,Z 296.905,A -85,B 0,C 180,E1 -9253.465,E2 -9253.465} C_VEL
LIN {X 0,Y 406.594,Z 302.848,A -85,B 0,C 180,E1 -9254.158,E2 -9254.158} C_VEL
LIN {X 0,Y 406.744,Z 321.177,A -85,B 0,C 180,E1 -9255.971,E2 -9255.971} C_VEL
LIN {X 0,Y 407.641,Z 325.401,A -85,B 0,C 180,E1 -9256.467,E2 -9256.467} C_VEL
LIN {X 0,Y 409.893,Z 332.99,A -85,B 0,C 180,E1 -9257.413,E2 -9257.413} C_VEL
LIN {X 0,Y 407.639,Z 375.156,A -85,B 0,C 180,E1 -9261.299,E2 -9261.299} C_VEL
LIN {X 0,Y 405.431,Z 415.192,A -85,B 0,C 180,E1 -9264.976,E2 -9264.976} C_VEL
LIN {X 0,Y 403.186,Z 457.574,A -85,B 0,C 180,E1 -9268.862,E2 -9268.862} C_VEL
LIN {X 0,Y 402.086,Z 479.024,A -85,B 0,C 180,E1 -9270.818,E2 -9270.818} C_VEL
LIN {X 0,Y 403.84,Z 496.079,A -85,B 0,C 180,E1 -9271.26,E2 -9271.26} C_VEL
LIN {X 0,Y 401.543,Z 622.324,A -85,B 0,C 180,E1 -9273.581,E2 -9273.581} C_VEL
LIN {X 0,Y 400.96,Z 638.334,A -85,B 0,C 180,E1 -9274.137,E2 -9274.137} C_VEL
LIN {X 0,Y 400.091,Z 653.927,A -85,B 0,C 180,E1 -9274.944,E2 -9274.944} C_VEL
LIN {X 0,Y 399.033,Z 668.365,A -85,B 0,C 180,E1 -9275.96,E2 -9275.96} C_VEL
LIN {X 0,Y 397.76,Z 682.856,A -85,B 0,C 180,E1 -9277.291,E2 -9277.291} C_VEL
LIN {X 0,Y 396.552,Z 695.298,A -85,B 0,C 180,E1 -9278.738,E2 -9278.738} C_VEL
LIN {X 0,Y 395.31,Z 707.279,A -85,B 0,C 180,E1 -9280.491,E2 -9280.491} C_VEL
LIN {X 0,Y 394.288,Z 717.193,A -85,B 0,C 180,E1 -9282.297,E2 -9282.297} C_VEL
LIN {X 0,Y 393.375,Z 726.397,A -85,B 0,C 180,E1 -9284.438,E2 -9284.438} C_VEL
LIN {X 0,Y 392.762,Z 733.47,A -85,B 0,C 180,E1 -9286.564,E2 -9286.564} C_VEL
LIN {X 0,Y 392.355,Z 739.072,A -85,B 0,C 180,E1 -9288.881,E2 -9288.881} C_VEL
LIN {X 0,Y 392.153,Z 742.883,A -85,B 0,C 180,E1 -9291.224,E2 -9291.224} C_VEL
LIN {X 0,Y 392.075,Z 744.872,A -85,B 0,C 180,E1 -9293.6,E2 -9293.6} C_VEL
LIN {X 0,Y 392.076,Z 745.149,A -85,B 0,C 180,E1 -9296.014,E2 -9296.014} C_VEL
LIN {X 0,Y 392.141,Z 743.583,A -85,B 0,C 180,E1 -9298.397,E2 -9298.397} C_VEL
LIN {X 0,Y 392.336,Z 740.201,A -85,B 0,C 180,E1 -9300.813,E2 -9300.813} C_VEL
LIN {X 0,Y 392.707,Z 735.085,A -85,B 0,C 180,E1 -9303.105,E2 -9303.105} C_VEL
LIN {X 0,Y 393.319,Z 728.311,A -85,B 0,C 180,E1 -9305.311,E2 -9305.311} C_VEL
